	12:	//MoveZ-Free ready? -> Piece zuordnen -> Action ready
		IF NOT pStampSupport^.M_GetActionBusy(E_Action.ACTION_MoveZ) THEN
			nActionState := 80;
			IF bTakePiece THEN
				//Piece von Magazin auf Support übertragen
				IF pStampSupport^.P_bStampInSupport THEN
					//das letze Slot ermitteln
					stError.ErrorId := fbObjectDirectory.M_MoveObject(pPiece,pStampSupport,pStampSupport^.P_nNumberOfSlots);
				ELSE //Take fehlgeschlagen, weil Stamp nicht im Support detektierbar
					stError.ErrorId := E_ErrorIdCmd.ERRORID_PieceExchangeFailed;
				END_IF
			ELSE //Drop
				//Piece von Support auf Magazin übertragen
				IF pStampSupport^.P_bStampInSupport THEN //Drop fehlgeschlagen, weil weil Stamp noch im Support detektierbar
					stError.ErrorId := E_ErrorIdCmd.ERRORID_PieceExchangeFailed;
					nActionState := 99;
				ELSE
					stError.ErrorId := fbObjectDirectory.M_MoveObject(pPiece,pTarget,pPieceSlot^.nNr);
				END_IF
			END_IF
			pPiece^.P_bIgnoreOffset := FALSE;
			IF stError.ErrorId > 0 THEN
				nActionState := 99;
			ELSE
				nActionState := 80;		
			END_IF
		END_IF
		
	70:	//Action abbrechen
		nActionState := 80;
		pPiece^.P_bIgnoreOffset := FALSE;
		IF fbMoveToTarget.bBusy THEN
			fbMoveToTarget(bStop:= TRUE);
			nActionState := 70;
		ELSIF pStampSupport^.M_GetActionBusy(E_Action.ACTION_MoveZ) THEN
			pStampSupport^.M_CancelAction(E_Action.ACTION_MoveZ);
			nActionState := 70;
		ELSE
			fbMoveToTarget(bExecute:= FALSE);
		END_IF
		
		IF pStampSupport^.M_GetActionBusy(E_Action.ACTION_LockUnlock) THEN
			pStampSupport^.M_CancelAction(E_Action.ACTION_LockUnlock);
			nActionState := 70;
		END_IF
		
		IF pStampSupport^.M_GetActionBusy(E_Action.ACTION_StampAdjust) THEN
			pStampSupport^.M_CancelAction(E_Action.ACTION_StampAdjust);
			nActionState := 70;
		END_IF
END_CASE

//Errorhandling
IF nActionState = 99 THEN
	pPiece^.P_bIgnoreOffset := FALSE;
	fbMoveToTarget(bExecute:= FALSE);
	stError.ObjectId := pStampSupport^.P_nObjectID;
	stError.Cmd := E_Action.ACTION_ExchangePiece;
	stError.POUAction := E_POUACT.POUACT_A_ExchangeStamp;
	fbErrorList.M_Add(stError);
END_IF
END_ACTION

ACTION A_ExchangeTip:
stError.POUState := nActionState;

IF pMzTool^.P_bError THEN
	stError.ErrorId := pMzTool^.P_nErrorId;
	nActionState := 99;
END_IF

IF pMzTool^.P_bCanceled AND nActionState > 0 AND nActionState < 70 THEN
	//MzTool wurde durch StopDevice abgebrochen
	nActionState := 70;
END_IF

CASE nActionState OF
	0:	//MoveToTarget auf Slot
		nActionState := 1;
		MEMSET(ADR(stActionData),0,SIZEOF(stActionData));
		stActionData.eAction := E_Action.ACTION_MoveToTarget;
		stActionData.nObject := pMzTool^.P_nObjectID;
		stActionData.nTarget := pTarget^.P_nObjectID;
		stActionData.aParams[1] := E_TargetRef.TARGETREF_Slot;
		stActionData.aParams[2] := pPieceSlot^.nNr;
		stActionData.aParams[3] := 0;
		stActionData.aParams[5] := -1;	//MaxSpeed X
		stActionData.aParams[6] := -1;	//MaxSpeed Y
		stActionData.aParams[7] := -1;	//MaxSpeed Z
		
		IF NOT bTakePiece THEN //Drop
			stDimension :=  pPiece^.P_stDimension;
			stActionData.aParams[10] := - REAL_TO_DINT(stDimension.Height - pPiece^.P_rZOverlapTool);
		END_IF
		
		pPiece^.P_bIgnoreOffset := TRUE;
		
		stError.ErrorId := fbMoveToTarget.M_SetAndCheckParams(stActionData);
		IF stError.ErrorId > 0 THEN	//Error
			nActionState := 99;
		ELSE
			fbMoveToTarget(bExecute:= TRUE);
			nActionState := 1;
		END_IF		
		
	1:	//MoveToTarget ready? -> MoveZ bei Take bzw Eject bei Drop
		fbMoveToTarget(bExecute:= TRUE);
		IF NOT fbMoveToTarget.bBusy THEN
			IF fbMoveToTarget.bError THEN
				stError.ErrorId := fbMoveToTarget.nErrorId;
				nActionState := 99;
			ELSE
				IF bTakePiece THEN //Take
					//Z-Zustellung um OverlapTool und SumDockOffset
					stActionData.eAction := E_Action.ACTION_MoveZ;
					stActionData.aParams[1] := E_MoveMode.MODE_Relative;
					stActionData.aParams[2] := REAL_TO_DINT(pPiece^.P_rZOverlapTool * -1 + rSumDockOffset);
					stActionData.aParams[3] := 4000; //MoveSpeed
				ELSE
					stActionData.eAction := E_Action.ACTION_Eject;
				END_IF
				stError.ErrorId := pMzTool^.M_ExeAction(stActionData);
				IF stError.ErrorId > 0 THEN	//Error
					nActionState := 99;
				ELSE
					nActionState := 2;
				END_IF		
			END_IF
			fbMoveToTarget(bExecute:= FALSE);
		END_IF
		
	2:	//MoveZ bzw Eject ready? -> MoveZ-Home
		IF NOT (pMzTool^.M_GetActionBusy(E_Action.ACTION_MoveZ) OR pMzTool^.M_GetActionBusy(E_Action.ACTION_Eject)) THEN
			nActionState := 3;
			MEMSET(ADR(stActionData),0,SIZEOF(stActionData));
			stActionData.eAction := E_Action.ACTION_MoveZ;
			stActionData.aParams[1] := E_MoveMode.MODE_Home;
			stActionData.aParams[3] := -1; //MoveSpeed
			stError.ErrorId := pMzTool^.M_ExeAction(stActionData);
			IF stError.ErrorId > 0 THEN	//Error
				nActionState := 99;
			END_IF
		END_IF
		
	3:	//MoveZ-Home ready -> Piece zuordnen -> Action ready
		IF NOT pMzTool^.M_GetActionBusy(E_Action.ACTION_MoveZ) THEN
			IF bTakePiece THEN
				//Piece von NeedleRack auf MzTool übertragen
				stError.ErrorId := fbObjectDirectory.M_MoveObject(pPiece,pMzTool,1);
			ELSE
				//Piece von MzTool auf Rack übertragen
				stError.ErrorId := fbObjectDirectory.M_MoveObject(pPiece,pTarget,pPieceSlot^.nNr);
				//Offset von Piece löschen
				stPoint1.X := 0;
				stPoint1.Y := 0;
				stPoint1.Z := 0;
				pPiece^.P_stOffset := stPoint1;
				//Tip als "used" kennzeichnen
				pTip := pPiece;
				pTip^.P_bUsed := TRUE;
				fbObjectDirectory.M_SetObjChange(pPiece^.P_nObjectID);
			END_IF
			pPiece^.P_bIgnoreOffset := FALSE;
			IF stError.ErrorId > 0 THEN
				nActionState := 99;
			ELSE
				nActionState := 80;		
			END_IF
		END_IF
 		
	70:	//Action abbrechen
		pPiece^.P_bIgnoreOffset := FALSE;
		IF fbMoveToTarget.bBusy THEN
			fbMoveToTarget(bStop:= TRUE);
		ELSIF pMzTool^.M_GetActionBusy(E_Action.ACTION_MoveZ) THEN
			pMzTool^.M_CancelAction(E_Action.ACTION_MoveZ);
		ELSE
			fbMoveToTarget(bExecute:= FALSE);
			nActionState := 80;
		END_IF		
END_CASE

//Errorhandling
IF nActionState = 99 THEN
	fbMoveToTarget(bExecute:= FALSE);
	pPiece^.P_bIgnoreOffset := FALSE;
	stError.ObjectId := pMzTool^.P_nObjectID;
	stError.Cmd := E_Action.ACTION_ExchangePiece;
	stError.POUAction := E_POUACT.POUACT_A_ExchangeTip;
	fbErrorList.M_Add(stError);
END_IF
END_ACTION

ACTION A_ExchangeVial:
stError.POUState := nActionState;

IF pMzTool^.P_bError THEN
	stError.ObjectId := pMzTool^.P_nObjectID;
	stError.ErrorId := pMzTool^.P_nErrorId;
	nActionState := 99;
ELSE
	IF pReactor > 0 THEN
		IF pReactor^.P_bError THEN
			stError.ObjectId := pReactor^.P_nObjectID;
			stError.ErrorId := pReactor^.P_nErrorId;
			nActionState := 99;
		END_IF
	END_IF	
END_IF

IF pMzTool^.P_bCanceled AND nActionState > 0 AND nActionState < 70 THEN
	//MzTool wurde durch StopDevice abgebrochen
	nActionState := 70;
END_IF

CASE nActionState OF
	0:	//Prepare
		//Druck
		//Reactor öffnen
		//Überprüfen, ob VialKlemme zu bzw prüfen, ob Vial im Slot
		//VialDetection
		nActionState := 5;
		timer1(IN:= FALSE);
		IF pTarget^.P_eObjectType = E_ObjectType.OBJECTTYPE_Reactor THEN
			pReactor := pTarget;
			MEMSET(ADR(stActionData),0,SIZEOF(stActionData));
			stActionData.eAction := E_Action.ACTION_DetectVial;
			stActionData.aParams[1] := E_OpClState.Open;
			
			stError.ErrorId := pReactor^.M_ExeAction(stActionData);
			IF stError.ErrorId > 0 THEN
				stError.ObjectId := pReactor^.P_nObjectID;
				nActionState := 99;
			ELSE
				nActionState := 1;	
			END_IF			
		END_IF
		
		IF nActionState <> 99 THEN
			//Hier kann die XY-Zustellung bereits angestoßen werden
			MEMSET(ADR(stActionData),0,SIZEOF(stActionData));
			//stActionData.bIntern := TRUE;
			stActionData.eAction := E_Action.ACTION_MoveToTarget;
			stActionData.nObject := pMzTool^.P_nObjectID;
			stActionData.nTarget := pTarget^.P_nObjectID;
			stActionData.aParams[1] := E_TargetRef.TARGETREF_Slot;
			stActionData.aParams[2] := pPieceSlot^.nNr;
			stActionData.aParams[3] := 0;
			stActionData.aParams[5] := -1;	//MaxSpeed X
			stActionData.aParams[6] := -1;	//MaxSpeed Y
			stActionData.aParams[7] := 0;	//MaxSpeed Z
			stError.ErrorId := fbMoveToTarget.M_SetAndCheckParams(stActionData);
			IF stError.ErrorId > 0 THEN	//Error
				stError.ObjectId := pMzTool^.P_nObjectID;
				nActionState := 99;
			ELSE
				IF pMzTool^.P_eObjectType = E_ObjectType.OBJECTTYPE_TriplePip THEN //PneuChannel vorbereiten
					pTriplePip := pMzTool;
					MEMSET(ADR(stActionData),0,SIZEOF(stActionData));
					stActionData.eAction := E_Action.ACTION_SetVacuum;
					IF bTakePiece THEN
						stActionData.aParams[1] := 1; //Fertigmeldung wenn Solldruck erreicht
						stActionData.aParams[2] := -80; //Value in kPa
						stActionData.aParams[3] := 5; //Toleranz
						stActionData.aParams[4] := 5; //Toleranz
						stActionData.aParams[5] := 10000; //Timeout in ms
						stError.ErrorId :=  pMzTool^.M_ExeAction(stActionData);
						IF stError.ErrorId > 0 THEN
							stError.ObjectId := pMzTool^.P_nObjectID;
							nActionState := 99;
						ELSE
							//Ventil aus falls noch an
							MEMSET(ADR(stActionData),0,SIZEOF(stActionData));
							stActionData.eAction := E_Action.ACTION_SwitchPressure;
							stActionData.aParams[1] := E_PressCtrl.PRESSCTRL_Off;
							stError.ErrorId := pMzTool^.M_ExeAction(stActionData);
							IF stError.ErrorId > 0 THEN
								stError.ObjectId := pMzTool^.P_nObjectID;
								nActionState := 99;
							ELSE
								nActionState := 1;
							END_IF
						END_IF
					ELSE
						nActionState := 1;
					END_IF
				END_IF				
			END_IF
		END_IF
		IF nActionState = 1 THEN
			fbMoveToTarget(bExecute:= TRUE);
		END_IF
 		
	1:	//Prepare ready?
		nActionState := 5;
		IF pTarget^.P_eObjectType = E_ObjectType.OBJECTTYPE_Reactor THEN
			nActionState := 2;
			IF pReactor^.M_GetActionBusy(E_Action.ACTION_DetectVial) THEN
				nActionState := 1;
			END_IF
		END_IF
		
		IF pMzTool^.P_eObjectType = E_ObjectType.OBJECTTYPE_TriplePip THEN //Vacuum OK?
			IF pMzTool^.M_GetActionBusy(E_Action.ACTION_SetVacuum) THEN
				nActionState := 1;
			END_IF
		END_IF
		
	2:	//Auswertung VialDetection
		nActionState := 3;
		IF bTakePiece THEN
			IF NOT pReactor^.P_bVialInSlot THEN
				stError.ErrorId := E_ErrorIdCmd.ERRORID_NoVialInReactor;
				nActionState := 99;
			END_IF
		ELSE
			IF pReactor^.P_bVialInSlot THEN
				stError.ErrorId := E_ErrorIdCmd.ERRORID_VialAlreadyInReactor;		
				nActionState := 99;
			END_IF
		END_IF
		
	3:	//Open Reactor
		nActionState := 4;
		MEMSET(ADR(stActionData),0,SIZEOF(stActionData));
		stActionData.eAction := E_Action.ACTION_ReactorOpCl;
		stActionData.aParams[1] := E_ReactDrive.CoverBoth;
		stActionData.aParams[2] := E_OpClCtrl.Open;
		stError.ErrorId := pReactor^.M_ExeAction(stActionData);
		IF stError.ErrorId > 0 THEN
			stError.ObjectId := pReactor^.P_nObjectID;
			nActionState := 99;
		END_IF			
		
	4:	//Reactor open?
		IF NOT pReactor^.M_GetActionBusy(E_Action.ACTION_ReactorOpCl) THEN
			nActionState := 5;
		END_IF
	
	5:	//MoveToTarget Slot
		fbMoveToTarget(bExecute:= TRUE);
		IF NOT fbMoveToTarget.bBusy THEN
			IF fbMoveToTarget.bError THEN
				stError.ErrorId := fbMoveToTarget.nErrorId;
				nActionState := 99;
				fbMoveToTarget(bExecute:= FALSE);
			ELSE
				MEMSET(ADR(stActionData),0,SIZEOF(stActionData));
				stActionData.eAction := E_Action.ACTION_MoveToTarget;
				stActionData.nObject := pMzTool^.P_nObjectID;
				stActionData.nTarget := pTarget^.P_nObjectID;
				stActionData.aParams[1] := E_TargetRef.TARGETREF_Slot;
				stActionData.aParams[2] := pPieceSlot^.nNr;
				stActionData.aParams[3] := 0;
				stActionData.aParams[5] := -1;	//MaxSpeed X
				stActionData.aParams[6] := -1;	//MaxSpeed Y
				stActionData.aParams[7] := -1;	//MaxSpeed Z
				IF bTakePiece THEN
					stActionData.aParams[10] := REAL_TO_DINT(rSumDockOffset);
				END_IF
				fbMoveToTarget(bExecute:= FALSE);
				stError.ErrorId := fbMoveToTarget.M_SetAndCheckParams(stActionData);
				IF stError.ErrorId > 0 THEN	//Error
					stError.ObjectId := pMzTool^.P_nObjectID;
					nActionState := 99;
				ELSE
					fbMoveToTarget(bExecute:= TRUE);
					nActionState := 6;
				END_IF
			END_IF
		END_IF
	
	6:	//MoveToTarget ready? -> Übergabe
		fbMoveToTarget(bExecute:= TRUE);
		IF NOT fbMoveToTarget.bBusy THEN
			IF fbMoveToTarget.bError THEN
				stError.ErrorId := fbMoveToTarget.nErrorId;
				nActionState := 99;
			ELSE
				IF bTakePiece THEN
					nActionState := 7;
				ELSE
					nActionState := 10;
				END_IF
			END_IF
			fbMoveToTarget(bExecute:= FALSE);
		END_IF
		
	7:	//Übergabe Take
		nActionState := 8;
		MEMSET(ADR(stActionData),0,SIZEOF(stActionData));
		stActionData.eAction := E_Action.ACTION_SwitchPressure;
		//Vacuum zuschalten
		stActionData.aParams[1] := E_PressCtrl.PRESSCTRL_VacOn;
		stError.ErrorId := pMzTool^.M_ExeAction(stActionData);
		IF stError.ErrorId > 0 THEN
			stError.ObjectId := pMzTool^.P_nObjectID;
			nActionState := 99;
		END_IF
		
	8:	//Zeit warten
		timer1(IN:= TRUE, PT:=T#1S);
		IF timer1.Q THEN
			timer1(IN:= FALSE);
			nActionState := 9;
		END_IF
		
	9:	//Vaccum OK ? -> MoveZ-Free
		IF pTriplePip^.M_GetVacuumOk(nSetPressValue:= pTriplePip^.P_nHoldVacVial, nSetPressTolPlus:= 0, nSetPressTolMin := 99) THEN
			nActionState := 13;
		END_IF
		
	10:	//Übergabe Drop
		//MoveZ relativ um Slot-Tiefe abzüglich 1mm
		nActionState := 11;
		MEMSET(ADR(stActionData),0,SIZEOF(stActionData));
		stActionData.eAction := E_Action.ACTION_MoveZ;
		stActionData.aParams[1] := E_MoveMode.MODE_Relative;
		stActionData.aParams[2] := -(REAL_TO_DINT((pPieceSlot^.P_rDepth - 1000)));
		stActionData.aParams[3] := 20000; //MoveSpeed
		stError.ErrorId := pMzTool^.M_ExeAction(stActionData);
		IF stError.ErrorId > 0 THEN	//Error
			stError.ObjectId := pMzTool^.P_nObjectID;
			nActionState := 99;
		END_IF
	
	11:	//MoveZ ready? -> MoveX 1mm zum lösen vom Vial, Vacuum Off
		IF NOT pMzTool^.M_GetActionBusy(E_Action.ACTION_MoveZ) THEN
			nActionState := 12;
			//Move 1mm in X, damit Vial sich vom Tool löst
			MEMSET(ADR(stActionData),0,SIZEOF(stActionData));
			stActionData.eAction := E_Action.ACTION_MoveX;
			stActionData.aParams[1] := E_MoveMode.MODE_Relative;
			stActionData.aParams[2] := 500;
			stActionData.aParams[3] := 10000; //MoveSpeed
			stActionData.aParams[4] := 1; //Ignore Collision
			stError.ErrorId := pMzTool^.M_ExeAction(stActionData);
			IF stError.ErrorId > 0 THEN	//Error
				stError.ObjectId := pMzTool^.P_nObjectID;
				nActionState := 99;
			ELSE
				//Vacuum OFF
				MEMSET(ADR(stActionData),0,SIZEOF(stActionData));
				stActionData.eAction := E_Action.ACTION_SwitchPressure;
				stActionData.aParams[1] := E_PressCtrl.PRESSCTRL_Off;
				stError.ErrorId :=  pMzTool^.M_ExeAction(stActionData);
				IF stError.ErrorId > 0 THEN
					stError.ObjectId := pMzTool^.P_nObjectID;
					nActionState := 99;
				ELSE
					//Set Vacuum "0"
					MEMSET(ADR(stActionData),0,SIZEOF(stActionData));
					stActionData.eAction := E_Action.ACTION_SetVacuum;
					stActionData.aParams[1] := 0; //Fertigmeldung sofort
					stActionData.aParams[2] := 0; //Value in kPa
					stError.ErrorId :=  pMzTool^.M_ExeAction(stActionData);
					IF stError.ErrorId > 0 THEN
						stError.ObjectId := pMzTool^.P_nObjectID;
						stError.POUState := nActionState;
						nActionState := 99;
					END_IF
				END_IF
			END_IF
		END_IF
		
	12:	//MoveX ready? -> MoveZ 1mm nach oben
		IF NOT pMzTool^.M_GetActionBusy(E_Action.ACTION_MoveX) THEN
			nActionState := 13;
			MEMSET(ADR(stActionData),0,SIZEOF(stActionData));
			stActionData.eAction := E_Action.ACTION_MoveZ;
			stActionData.aParams[1] := E_MoveMode.MODE_Relative;
			stActionData.aParams[2] := 500; //0,5mm nach oben
			stActionData.aParams[3] := 1000; //MoveSpeed
			stError.ErrorId :=  pMzTool^.M_ExeAction(stActionData);
			IF stError.ErrorId > 0 THEN
				stError.ObjectId := pMzTool^.P_nObjectID;
				nActionState := 99;
			END_IF
		END_IF
		
	13:	//MoveZ-Free
		IF NOT pMzTool^.M_GetActionBusy(E_Action.ACTION_MoveZ) THEN
			MEMSET(ADR(stActionData),0,SIZEOF(stActionData));
			stActionData.eAction := E_Action.ACTION_MoveZ;
			stActionData.aParams[1] := E_MoveMode.MODE_Home;
			stActionData.aParams[3] := -1; //MoveSpeed
			stError.ErrorId := pMzTool^.M_ExeAction(stActionData);
			IF stError.ErrorId > 0 THEN	//Error
				stError.ObjectId := pMzTool^.P_nObjectID;
				nActionState := 99;
			END_IF
			nActionState := 14;
		END_IF

	14:	//MoveZ-Free ready? -> Action ready
		IF NOT pMzTool^.M_GetActionBusy(E_Action.ACTION_MoveZ) THEN
			IF bTakePiece THEN	//Vial von Target auf MzTool übertragen
				stError.ErrorId := fbObjectDirectory.M_MoveObject(pPiece,pMzTool,1);
				pVial := pPiece;
				pVial^.P_bUsed := TRUE;
				fbObjectDirectory.M_SetObjChange(pPiece^.P_nObjectID);
			ELSE	//Vial von MzTool auf Target übertragen
				stError.ErrorId := fbObjectDirectory.M_MoveObject(pPiece,pTarget,pPieceSlot^.nNr);
			END_IF
			IF stError.ErrorId > 0 THEN
				nActionState := 99;
			ELSE
				nActionState := 80;		
			END_IF
		END_IF
		
	70:	//Abbrechen
		IF NOT bTakePiece THEN
			nActionState := 71;
		ELSE
			nActionState := 80;
		END_IF
	
		IF fbMoveToTarget.bBusy THEN
			fbMoveToTarget(bStop:= TRUE);
			nActionState := 70;
		ELSIF pMzTool^.M_GetActionBusy(E_Action.ACTION_MoveX) THEN
			pMzTool^.M_CancelAction(E_Action.ACTION_MoveX);
			nActionState := 70;
		ELSIF pMzTool^.M_GetActionBusy(E_Action.ACTION_MoveZ) THEN
			pMzTool^.M_CancelAction(E_Action.ACTION_MoveZ);
			nActionState := 70;
		END_IF
		
		IF pMzTool^.M_GetActionBusy(E_Action.ACTION_SetVacuum) THEN
			nActionState := 70;
			pMzTool^.M_CancelAction(E_Action.ACTION_SetVacuum);
		END_IF
		
		IF pMzTool^.M_GetActionBusy(E_Action.ACTION_SwitchPressure) THEN
			nActionState := 70;
			pMzTool^.M_CancelAction(E_Action.ACTION_SwitchPressure);
		END_IF
		
		IF pReactor > 0 THEN
			IF pReactor^.M_GetActionBusy(E_action.ACTION_ReactorOpCl) THEN
				pReactor^.M_CancelAction(E_action.ACTION_ReactorOpCl);
				nActionState := 70;
			ELSIF pReactor^.M_GetActionBusy(E_action.ACTION_DetectVial) THEN
				pReactor^.M_CancelAction(E_action.ACTION_DetectVial);
				nActionState := 70;
			END_IF
		END_IF	
	
	71:	//Vacuum OFF (nur wenn Take)
		nActionState := 80;
		stActionData.eAction := E_Action.ACTION_SwitchPressure;
		stActionData.aParams[1] := E_PressCtrl.PRESSCTRL_Off;
		stError.ErrorId := pMzTool^.M_ExeAction(stActionData);
		IF stError.ErrorId = 0 THEN
			stActionData.eAction := E_Action.ACTION_SetVacuum;
			stActionData.aParams[1] := 0; //Sofortige Fertigmeldung
			stActionData.aParams[2] := 0; //Druck
			stError.ErrorId := pMzTool^.M_ExeAction(stActionData);
			IF stError.ErrorId > 0 THEN
				stError.ObjectId := pMzTool^.P_nObjectID;
				nActionState := 99;
			END_IF
		END_IF	
END_CASE

//Errorhandling
IF nActionState = 99 THEN
	IF bTakePiece THEN
		stActionData.eAction := E_Action.ACTION_SwitchPressure;
		stActionData.aParams[1] := E_PressCtrl.PRESSCTRL_Off;
		pMzTool^.M_ExeAction(stActionData);
		stActionData.eAction := E_Action.ACTION_SetVacuum;
		stActionData.aParams[1] := 0; //Sofortige Fertigmeldung
		stActionData.aParams[2] := 0; //Druck
		pMzTool^.M_ExeAction(stActionData);
	END_IF
	pPiece^.P_bIgnoreOffset := FALSE;
	fbMoveToTarget(bExecute:= FALSE);
	stError.ObjectId := pMzTool^.P_nObjectID;
	stError.Cmd := E_Action.ACTION_ExchangePiece;
	stError.POUAction := E_POUACT.POUACT_A_ExchangeVial;
	fbErrorList.M_Add(stError);
END_IF
END_ACTION

ACTION A_ExchangeVialGripper:
stError.POUState := nActionState;

IF pMzTool^.P_bError THEN
	stError.ObjectId := pMzTool^.P_nObjectID;
	stError.ErrorId := pMzTool^.P_nErrorId;
	nActionState := 99;
ELSE
	IF pPowderStation > 0 AND_THEN pTarget = pPowderStation THEN
		IF pPowderStation^.P_bError THEN
			stError.ObjectId := pPowderStation^.P_nObjectID;
			stError.ErrorId := pPowderStation^.P_nErrorId;
			nActionState := 99;
		END_IF
	ELSIF pReactor > 0 AND_THEN pTarget = pReactor THEN
		IF pReactor^.P_bError THEN
			stError.ObjectId := pReactor^.P_nObjectID;
			stError.ErrorId := pReactor^.P_nErrorId;
			nActionState := 99;
		END_IF
	END_IF
END_IF

IF pMzTool^.P_bCanceled AND nActionState > 0 AND nActionState < 70 THEN
	//MzTool wurde durch StopDevice abgebrochen
	nActionState := 70;
END_IF

CASE nActionState OF
	0:	//Move free für Gripper-Test
		MEMSET(ADR(stActionData),0,SIZEOF(stActionData));
		stActionData.eAction := E_Action.ACTION_MoveZ;
		stActionData.aParams[1] := E_MoveMode.MODE_Home;
		stActionData.aParams[3] := -1; //MoveSpeed
		stError.ErrorId := pMzTool^.M_ExeAction(stActionData);
		IF stError.ErrorId > 0 THEN	//Error
			stError.ObjectId := pMzTool^.P_nObjectID;
			nActionState := 99;
		ELSE
			nActionState := 1;
		END_IF
		
	1:	//Move free ready?
		IF NOT pMzTool^.M_GetActionBusy(E_Action.ACTION_MoveZ) THEN
			//Gripper vorbereiten bzw. checken, ob State zur Belegung des VialSlots passt.
			//Auch bei TakePiece muss zuerst geschlosse werden, da ja aus irgendwelchen Gründen
			//noch ein Vial im Greifer sein kann und das Vial womöglich auf die Workplate falle würde
			stError.ErrorId := pGripper^.M_OpenClose(E_OpClCtrl.Close, FALSE);
			IF stError.ErrorId = 0 THEN
				nActionState := 2;
			ELSE
				nActionState := 99;
			END_IF			
		END_IF
	
	2:	//Gripper ready?
		IF NOT pGripper^.M_GetActionBusy(E_Action.ACTION_OpenClose) THEN
			IF bTakePiece THEN
				//Muss vollständig geschlossen sein, was bedeutet, dass sich kein Vial im Gripper befindet
				IF pGripper^.P_eCurrentGripperState = E_GripperState.FullyClosed THEN
					//wieder öffnen
					stError.ErrorId := pGripper^.M_OpenClose(E_OpClCtrl.Open, FALSE);
					IF stError.ErrorId = 0 THEN
						nActionState := 3;
					ELSE
						nActionState := 99;	
					END_IF
				ELSE
					stError.ErrorId := E_ErrorIdCmd.ERRORID_ToolNotFreeOrBlocked;
					nActionState := 99;
				END_IF
			ELSE //Drop
				IF pGripper^.P_eCurrentGripperState = E_GripperState.HalfClosed THEN
					IF pTarget^.P_eObjectType = E_ObjectType.OBJECTTYPE_PowderStation THEN
						nActionState := 10;
					 	
					ELSIF pTarget^.P_eObjectType = E_ObjectType.OBJECTTYPE_Reactor THEN
						nActionState := 20;
					ELSE
						nActionState := 30;
					END_IF
				ELSE
					stError.ErrorId := E_ErrorIdCmd.ERRORID_NoPieceOnTool;
					nActionState := 99;
				END_IF
			END_IF
		END_IF
		
	3:	//Gripper ready?
		IF NOT pGripper^.M_GetActionBusy(E_Action.ACTION_OpenClose) THEN
			IF pGripper^.P_eCurrentGripperState = E_GripperState.Open THEN
				IF pTarget^.P_eObjectType = E_ObjectType.OBJECTTYPE_PowderStation THEN
					nActionState := 10;
				ELSIF pTarget^.P_eObjectType = E_ObjectType.OBJECTTYPE_Reactor THEN
					nActionState := 20;
				ELSE
					nActionState := 30;
				END_IF
 			ELSE
				stError.ErrorId := E_ErrorIdCmd.ERRORID_CouldNotOpenGripper;
				nActionState := 99;
			END_IF
		END_IF
		
	10:	//PowderStation in ReloadPos fahren
		stActionData.eAction := E_Action.ACTION_PowdStatReload;
		stError.ErrorId := pPowderStation^.M_ExeAction(stActionData);
		IF stError.ErrorId > 0 THEN	//Error
			stError.ObjectId := pPowderStation^.P_nObjectID;
			nActionState := 99;
		ELSE
			nActionState := 11;
		END_IF
		
	11:	//RealoadPos ready?
		IF NOT pPowderStation^.M_GetActionBusy(E_Action.ACTION_PowdStatReload) THEN
			nActionState := 30;
		END_IF
		
	20: //Reaktor ist noch nicht implementiert
		stError.ErrorId := E_ErrorIdCmd.ERRORID_InvalidTarget;
		nActionState := 99;
		
	30:	//Wenn Drop, dann muss noch über den Vialdetector überprüft werden,
		//ob nicht schon ein Vial im Target steckt. Dazu muss also ein MoveToTarget
		//mit entsprechendem Offset gemacht werden.
		IF bTakePiece THEN
			nActionState := 32;
		ELSE
			//move zur Übergabe mit Offset und checken
			MEMSET(ADR(stActionData),0,SIZEOF(stActionData));
			stActionData.eAction := E_Action.ACTION_MoveToTarget;
			stActionData.nObject := pMzTool^.P_nObjectID;
			stActionData.nTarget := pTarget^.P_nObjectID;
			stActionData.aParams[1] := E_TargetRef.TARGETREF_Slot;
			stActionData.aParams[2] := pPieceSlot^.nNr;
			stActionData.aParams[3] := 0;
			stActionData.aParams[5] := -1;	//MaxSpeed X
			stActionData.aParams[6] := -1;	//MaxSpeed Y
			stActionData.aParams[7] := -1;	//MaxSpeed Z
			stActionData.aParams[8] :=	0;	//Offset X
			stActionData.aParams[9] :=	-25500;	//Offset Y
			stActionData.aParams[10] :=	15000;	//Offset Z	
			stError.ErrorId := fbMoveToTarget.M_SetAndCheckParams(stActionData);
			IF stError.ErrorId > 0 THEN	//Error
				stError.ObjectId := pMzTool^.P_nObjectID;
				nActionState := 99;
			ELSE
				fbMoveToTarget(bExecute:= TRUE);
				nActionState := 31;
			END_IF
		END_IF
	
	31:	//MoveToTarget ready?
		fbMoveToTarget();
		IF NOT fbMoveToTarget.bBusy THEN
			IF fbMoveToTarget.bError THEN
				stError.ErrorId := fbMoveToTarget.nErrorId;
				nActionState := 99;
			ELSE
				IF NOT pGripper^.P_bVialDetector THEN //Es befindet sich ein Vial im Target
					stError.ErrorId := E_ErrorIdCmd.ERRORID_PieceAlreadyInSlot;
					nActionState := 99;
				ELSE
					//Eigentlicher MoveToTarget
					nActionState := 32;
				END_IF
			END_IF
			fbMoveToTarget(bExecute:= FALSE);
		END_IF
		
	32:	//MoveToTarget
		MEMSET(ADR(stActionData),0,SIZEOF(stActionData));
		stActionData.eAction := E_Action.ACTION_MoveToTarget;
		stActionData.nObject := pMzTool^.P_nObjectID;
		stActionData.nTarget := pTarget^.P_nObjectID;
		stActionData.aParams[1] := E_TargetRef.TARGETREF_Slot;
		stActionData.aParams[2] := pPieceSlot^.nNr;
		stActionData.aParams[3] := 0;
		stActionData.aParams[5] := -1;	//MaxSpeed X
		stActionData.aParams[6] := -1;	//MaxSpeed Y
		stActionData.aParams[7] := 30000;	//Speed Z
		IF bTakePiece THEN
			stActionData.aParams[10] := -REAL_TO_DINT(pPiece^.P_rZOverlapTool);
		END_IF
		
		stError.ErrorId := fbMoveToTarget.M_SetAndCheckParams(stActionData);
		IF stError.ErrorId > 0 THEN	//Error
			stError.ObjectId := pMzTool^.P_nObjectID;
			nActionState := 99;
		ELSE
			fbMoveToTarget(bExecute:= TRUE);
			nActionState := 33;
		END_IF
	
	33:	//MoveToTarget ready?
		fbMoveToTarget();
		IF NOT fbMoveToTarget.bBusy THEN
			IF fbMoveToTarget.bError THEN
				stError.ErrorId := fbMoveToTarget.nErrorId;
				nActionState := 99;
			ELSE
				IF bTakePiece THEN
					nActionState := 40;
				ELSE //Drop
					nActionState := 42;
				END_IF
			END_IF
			fbMoveToTarget(bExecute:= FALSE);
		END_IF
		
	40:	//Übergabe Take -> Close Gripper
		stError.ErrorId := pGripper^.M_OpenClose(E_OpClCtrl.Close, FALSE);
		IF stError.ErrorId > 0 THEN
			nActionState := 99;
		ELSE
			nActionState := 41;
		END_IF
		
	41:	//Gripper closed? (HALF)
		IF NOT pGripper^.M_GetActionBusy(E_Action.ACTION_OpenClose) THEN
			IF pGripper^.P_eCurrentGripperState = E_GripperState.HalfClosed THEN
				nActionState := 50; //Move free
			ELSE
				stError.ErrorId := E_ErrorIdCmd.ERRORID_NoPieceTaken;
				nActionState := 99;
			END_IF
		END_IF
		
	42:	//Übergabe Drop ->MoveZ relativ um Slot-Tiefe abzüglich 1mm
		MEMSET(ADR(stActionData),0,SIZEOF(stActionData));
		stActionData.eAction := E_Action.ACTION_MoveZ;
		stActionData.aParams[1] := E_MoveMode.MODE_Relative;
		stActionData.aParams[2] := -(REAL_TO_DINT((pPieceSlot^.P_rDepth - 1000)));
		stActionData.aParams[3] := 20000; //MoveSpeed
		stError.ErrorId := pMzTool^.M_ExeAction(stActionData);
		IF stError.ErrorId > 0 THEN	//Error
			stError.ObjectId := pMzTool^.P_nObjectID;
			nActionState := 99;
		ELSE
			nActionState := 43;
		END_IF
		
	43: //MoveZ ready? -> Open Gripper
		IF NOT pMzTool^.M_GetActionBusy(E_Action.ACTION_MoveZ) THEN
			stError.ErrorId := pGripper^.M_OpenClose(E_OpClCtrl.Open, FALSE);
			IF stError.ErrorId > 0 THEN
				nActionState := 99;
			ELSE
				nActionState := 44;
			END_IF
		END_IF
		
	44:	//Gripper open?
		IF NOT pGripper^.M_GetActionBusy(E_Action.ACTION_OpenClose) THEN
			IF pGripper^.P_eCurrentGripperState = E_GripperState.Open THEN
				nActionState := 50; //Move free
			ELSE
				stError.ErrorId := E_ErrorIdCmd.ERRORID_NotFullyOpened;
				nActionState := 99;
			END_IF
		END_IF
		
	50:	//Move free
		MEMSET(ADR(stActionData),0,SIZEOF(stActionData));
		stActionData.eAction := E_Action.ACTION_MoveZ;
		stActionData.aParams[1] := E_MoveMode.MODE_Home;
		stActionData.aParams[3] := -1; //MoveSpeed
		stError.ErrorId := pMzTool^.M_ExeAction(stActionData);
		IF stError.ErrorId > 0 THEN	//Error
			stError.ObjectId := pMzTool^.P_nObjectID;
			nActionState := 99;
		ELSE
			nActionState := 51;
		END_IF
		
	51:	//MoveZ-Free ready? -> Action ready
		IF NOT pMzTool^.M_GetActionBusy(E_Action.ACTION_MoveZ) THEN
			//Vial richtig angekommen? Geht nur bei Gripper, Reaktor oder bei PowderStation
			IF bTakePiece THEN
				IF pGripper^.P_eCurrentGripperState = E_GripperState.HalfClosed THEN
					nActionState := 60; //weiter zu Vial im OD verschieben
				ELSE
					stError.ErrorId := E_ErrorIdCmd.ERRORID_NoPieceTaken;
					nActionState := 99;
				END_IF
			ELSE //Drop
				IF pTarget^.P_eObjectType = E_ObjectType.OBJECTTYPE_Reactor THEN
					//Hier muss die DetectAction noch ausgeführt werden
					MEMSET(ADR(stActionData),0,SIZEOF(stActionData));
					stActionData.eAction := E_Action.ACTION_DetectVial;
					stActionData.aParams[1] := E_OpClState.Closed;
					stError.ErrorId := pReactor^.M_ExeAction(stActionData);
					IF stError.ErrorId > 0 THEN
						stError.ObjectId := pReactor^.P_nObjectID;
						nActionState := 99;
					ELSE
						//nActionState := 15; //Überprüfung, ob Vial auch im Reaktor angekommen???
					END_IF
				ELSE
					nActionState := 60; //weiter zu Vial im OD verschieben
				END_IF
			END_IF
		END_IF
		
	60:	//Vial im OD verschieben
		IF bTakePiece THEN	//Vial von Target auf MzTool übertragen
			stError.ErrorId := fbObjectDirectory.M_MoveObject(pPiece,pMzTool,1);
			pVial := pPiece;
			//pVial^.P_bUsed := TRUE;
			fbObjectDirectory.M_SetObjChange(pPiece^.P_nObjectID);
		ELSE	//Vial von MzTool auf Target übertragen
			stError.ErrorId := fbObjectDirectory.M_MoveObject(pPiece,pTarget,pPieceSlot^.nNr);
		END_IF
		IF stError.ErrorId > 0 THEN
			nActionState := 99;
		ELSE
			nActionState := 80;		
		END_IF
	
	70:	//Abbrechen
		nActionState := 80;
		
		IF fbMoveToTarget.bBusy THEN
			fbMoveToTarget(bStop:= TRUE);
			nActionState := 70;
		ELSIF pMzTool^.M_GetActionBusy(E_Action.ACTION_MoveX) THEN
			pMzTool^.M_CancelAction(E_Action.ACTION_MoveX);
			nActionState := 70;
		ELSIF pMzTool^.M_GetActionBusy(E_Action.ACTION_MoveZ) THEN
			pMzTool^.M_CancelAction(E_Action.ACTION_MoveZ);
			nActionState := 70;
		END_IF
		
		IF pReactor > 0 THEN
			IF pReactor^.M_GetActionBusy(E_action.ACTION_ReactorOpCl) THEN
				pReactor^.M_CancelAction(E_action.ACTION_ReactorOpCl);
				nActionState := 70;
			ELSIF pReactor^.M_GetActionBusy(E_action.ACTION_DetectVial) THEN
				pReactor^.M_CancelAction(E_action.ACTION_DetectVial);
				nActionState := 70;
			END_IF
		END_IF	

END_CASE

//Errorhandling
IF nActionState = 99 THEN
	pPiece^.P_bIgnoreOffset := FALSE;
	fbMoveToTarget(bExecute:= FALSE);
	stError.ObjectId := pMzTool^.P_nObjectID;
	stError.Cmd := E_Action.ACTION_ExchangePiece;
	stError.POUAction := E_POUACT.POUACT_A_ExchangeVialGripper;
	fbErrorList.M_Add(stError);
END_IF
END_ACTION

ACTION A_GetPipSample:
stError.POUState := nActionState;

IF pMzTool^.P_bError THEN
	stError.ObjectId := pMzTool^.P_nObjectID;
	stError.ErrorId := pMzTool^.P_nErrorId;
	nActionState := 99;
END_IF

IF pMzTool^.P_bCanceled AND nActionState > 0 AND nActionState < 70 THEN
	//MzTool wurde durch StopDevice abgebrochen
	nActionState := 70;
END_IF

CASE nActionState OF
	0:	//MoveToTarget zu Mtp in PrePos
		timer1(IN:= FALSE);
		MEMSET(ADR(stActionData),0,SIZEOF(stActionData));
		stActionData.eAction := E_Action.ACTION_MoveToTarget;
		IF pMzTool^.P_eObjectType = E_ObjectType.OBJECTTYPE_TwinPiezoHolder THEN
			stActionData.nObject := pTwinPiezoHolder^.P_pPiezoPipFirst^.P_nObjectID;
		ELSE
			stActionData.nObject := pMzTool^.P_nObjectID;	
		END_IF
		stActionData.nTarget := pMtp^.P_nObjectID;
		stActionData.aParams[1] := E_TargetRef.TARGETREF_TwoDimArray;
		stActionData.aParams[2] := nCol;
		stActionData.aParams[3] := nRow;
		stActionData.aParams[5] := -1;	//MaxSpeed X
		stActionData.aParams[6] := -1;	//MaxSpeed Y
		stActionData.aParams[7] := -1;	//MaxSpeed Z
		stError.ErrorId := fbMoveToTarget.M_SetAndCheckParams(stActionData);
		IF stError.ErrorId > 0 THEN
			stError.ObjectId := pMzTool^.P_nObjectID;
			nActionState := 99;
		ELSE
			fbMoveToTarget(bExecute:= TRUE);
			nActionState := 1;
		END_IF
		
	1:	//MoveToTarget ready?
		fbMoveToTarget(bExecute:= TRUE);
		IF NOT fbMoveToTarget.bBusy THEN
			IF fbMoveToTarget.bError THEN
				stError.ErrorId := fbMoveToTarget.nErrorId;
				nActionState := 99;
			ELSE
				IF nQuantity2 > 0 THEN //AirGap
					MEMSET(ADR(stActionData),0,SIZEOF(stActionData));
					stActionData.eAction := E_Action.ACTION_Aspirate;
					stActionData.aParams[1] := nQuantity2; //Quantity Airgap
					stActionData.aParams[2] := nFlow1;
					stError.ErrorId := pMzTool^.M_ExeAction(stActionData);
					IF stError.ErrorId > 0 THEN
						nActionState := 99;
					ELSE
						nActionState := 2;
					END_IF
				ELSE
					nActionState := 4;
				END_IF
			END_IF
			fbMoveToTarget(bExecute:= FALSE);
		END_IF	
		
	2: //AirGap ready?
		IF NOT pMzTool^.M_GetActionBusy(E_Action.ACTION_Aspirate) THEN
			IF nTime > 0 THEN
				timer1(IN:= TRUE, PT:= DWORD_TO_TIME(nTime));
				nActionState := 3;
			ELSE
				nActionState := 4;
			END_IF
		END_IF
		
	3:	//Delay elapsed?
		timer1();
		IF timer1.Q THEN
			timer1(IN:= FALSE);
			nActionState := 4;
		END_IF
	
	4:	//Eintauchen in Well
		stPoint1 := pMtp^.M_GetAbsPos(pChildPos:= 0, eTargetRef:= E_TargetRef.TARGETREF_TwoDimArray, nParam1:= nCol, nParam2:= nRow,
									nParam3:= 1,nZLevel:= 1);			
		MEMSET(ADR(stActionData),0,SIZEOF(stActionData));
		stActionData.eAction := E_Action.ACTION_MoveZ;
		stActionData.aParams[1] := E_MoveMode.MODE_AbsWithOffset;
		stActionData.aParams[2] := REAL_TO_DINT(stPoint1.Z);
		stActionData.aParams[3] := -1;
		stError.ErrorId := pMzTool^.M_ExeAction(stActionData);
		IF stError.ErrorId > 0 THEN
			stError.ObjectId := pMzTool^.P_nObjectID;
			nActionState := 99;
		ELSE
			nActionState := 5;	
		END_IF
		
	5:	//Eintauchen ready? -> Aspirieren
		IF NOT pMzTool^.M_GetActionBusy(E_Action.ACTION_MoveZ) THEN
			nActionState := 6;
			MEMSET(ADR(stActionData),0,SIZEOF(stActionData));
			stActionData.eAction := E_Action.ACTION_Aspirate;
			stActionData.aParams[1] := nQuantity1;
			stActionData.aParams[2] := nFlow1;
			stError.ErrorId := pMzTool^.M_ExeAction(stActionData);
			IF stError.ErrorId > 0 THEN
				stError.ObjectId := pMzTool^.P_nObjectID;
				stError.POUState := nActionState;
				nActionState := 99;
			ELSE
				IF bGetPipSample_ActivatePiezo THEN
					MEMSET(ADR(stActionData),0,SIZEOF(stActionData));
					stActionData.eAction := E_Action.ACTION_DispenseDrops;
					stActionData.aParams[2] := 1; //Ein
					stActionData.aParams[5] := 1; //Skip valve move
					pMzTool^.M_ExeAction(stActionData);
				END_IF
			END_IF
		END_IF
		
	6:	//Aspirate ready? -> Delay
		IF NOT pMzTool^.M_GetActionBusy(E_Action.ACTION_Aspirate) THEN
			IF nTime > 0 THEN
				timer1(IN:= TRUE, PT:= DWORD_TO_TIME(nTime));
				nActionState := 7;
			ELSE
				nActionState := 8;
			END_IF
		END_IF
	
	7:	//Delay elapsed? -> bei Piezo au Bypass sonst MoveZ_Free
		timer1();
		IF timer1.Q THEN
			timer1(IN:= FALSE);
			IF pMzTool^.P_eObjectType = E_ObjectType.OBJECTTYPE_PiezoPip THEN
				nActionState := 8;
			ELSE
				nActionState := 10;
			END_IF
		END_IF
		
	8:	//Valve auf Bypass stellen
		IF bGetPipSample_SwitchBypass THEN
			MEMSET(ADR(stActionData),0,SIZEOF(stActionData));
			stActionData.eAction := E_Action.ACTION_DilMoveValve;
			stActionData.aParams[1] := 3; //Bypass-Position
			stError.ErrorId := pMzTool^.M_ExeAction(stActionData);
			IF stError.ErrorId > 0 THEN
				nActionState := 99;
			ELSE
				nActionState := 9;	
			END_IF		
		ELSE
			nActionState := 10;
		END_IF
		
	9:	//Valve auf Bypass?
		IF NOT pMzTool^.M_GetActionBusy(E_Action.ACTION_DilMoveValve) THEN
			nActionState := 10;
		END_IF
	
	10:	//MoveZ-Free
		pMzTool^.M_CancelAction(E_Action.ACTION_DispenseDrops);
		MEMSET(ADR(stActionData),0,SIZEOF(stActionData));
		stActionData.eAction := E_Action.ACTION_MoveZ;
		stActionData.aParams[1] := E_MoveMode.MODE_Free;
		stActionData.aParams[3] := -1; //MaxSpeed Z
		stError.ErrorId := pMzTool^.M_ExeAction(stActionData);
		IF stError.ErrorId > 0 THEN
			stError.ObjectId := pMzTool^.P_nObjectID;
			nActionState := 99;
		ELSE
			nActionState := 11;
		END_IF
		
	11:	//MoveZ-Free ready?
		IF NOT pMzTool^.M_GetActionBusy(E_Action.ACTION_MoveZ) THEN
			nActionState := 80;
 		END_IF
		
	70:	//Abbrechen
		nActionState := 80;
		IF fbMoveToTarget.bBusy THEN
			fbMoveToTarget(bStop:= TRUE);
			nActionState := 70;
		ELSIF pMzTool^.M_GetActionBusy(E_Action.ACTION_MoveZ) THEN
			pMzTool^.M_CancelAction(E_Action.ACTION_MoveZ);
			nActionState := 70;
		ELSE
			fbMoveToTarget(bExecute := FALSE);
		END_IF
		
		IF pMzTool^.M_GetActionBusy(E_Action.ACTION_Aspirate) THEN
			pMzTool^.M_CancelAction(E_Action.ACTION_Aspirate);
			nActionState := 70;
		END_IF
		
		IF pMzTool^.M_GetActionBusy(E_Action.ACTION_DilMoveValve) THEN
			pMzTool^.M_CancelAction(E_Action.ACTION_DilMoveValve);
			nActionState := 70;
		END_IF
END_CASE

//Errorhandling
IF nActionState = 99 THEN
	fbMoveToTarget(bExecute:= FALSE);
	stError.Cmd := E_Action.ACTION_GetPipSample;
	stError.ObjectId := pMzTool^.P_nObjectID;
	stError.POUAction := E_POUACT.POUACT_A_GetPipSample;
	fbErrorList.M_Add(stError);
END_IF
END_ACTION

ACTION A_InsertTool:
stError.POUState := nActionState;

IF pMzTool^.P_bError THEN
	stError.ErrorId := pMzTool^.P_nErrorId;
	nActionState := 99;
END_IF

IF pMzTool^.P_bCanceled AND nActionState > 0 AND nActionState < 70 THEN
	//MzTool wurde durch StopDevice abgebrochen
	nActionState := 70;
END_IF

CASE nActionState OF
	0:	//MoveToTarget auf Slot
		//Wenn aktuelle XY-Position des Tools mit der Position des Slots übereinstimmt(Tolerenz +-5µm)
		//muss kann MoveToTarget übersprungen werden
		//Hilfreich beim Anheben der Needle auf anderes Level ohne dass vorher herausgezogen wird
		stPoint1 := pMzTool^.P_stCurrentPosPhys;
		stPoint2 := pTarget^.M_GetAbsPos(pChildPos:= 0, eTargetRef,nTargetCol,nTargetRow,0,0);
		IF ABS(stPoint1.X - stPoint2.X) <= 5.0 AND ABS(stPoint1.Y - stPoint2.Y) <= 5.0 THEN
			nActionState := 3; //-> EIntauchen
			RETURN;
		END_IF
 		
		MEMSET(ADR(stActionData),0,SIZEOF(stActionData));
		stActionData.eAction := E_Action.ACTION_MoveToTarget;
		stActionData.nObject := pMzTool^.P_nObjectID;
		stActionData.nTarget := pTarget^.P_nObjectID;
		stActionData.aParams[1] := eTargetRef;
		stActionData.aParams[2] := nTargetCol;
		stActionData.aParams[3] := nTargetRow;
		stActionData.aParams[5] := -1;	//MaxSpeed X
		stActionData.aParams[6] := -1;	//MaxSpeed Y
		stActionData.aParams[7] := -1;	//MaxSpeed Z
		IF pTarget^.P_eObjectType = E_ObjectType.OBJECTTYPE_FlipTubeRack THEN
			stActionData.aParams[8] := -4000;	//XOffset	
			stActionData.aParams[10] := 1000;	//ZOffset	
		END_IF
		
		stError.ErrorId := fbMoveToTarget.M_SetAndCheckParams(stActionData);
		IF stError.ErrorId > 0 THEN	//Error
			nActionState := 99;
		ELSE
			fbMoveToTarget(bExecute:= TRUE);
			nActionState := 1;
		END_IF		
		
	1:	//MoveToTarget ready? (nur für FlipTube) (Deckel etwas weiter öffnen) MoveX
		fbMoveToTarget(bExecute:= TRUE);
		IF NOT fbMoveToTarget.bBusy THEN
			IF fbMoveToTarget.bError THEN
				stError.ErrorId := fbMoveToTarget.nErrorId;
				nActionState := 99;
			ELSE
				IF pTarget^.P_eObjectType = E_ObjectType.OBJECTTYPE_FlipTubeRack THEN //MoveX (Deckel öffnen)
					MEMSET(ADR(stActionData),0,SIZEOF(stActionData));
					stActionData.eAction := E_Action.ACTION_MoveX;
					stActionData.aParams[1] := E_MoveMode.MODE_Relative;
					stActionData.aParams[2] := 13000;
					stActionData.aParams[3] := 45000;
					stActionData.aParams[4] := 1;
					stError.ErrorId := pMzTool^.M_ExeAction(stActionData);
					IF stError.ErrorId > 0 THEN	//Error
						nActionState := 99;
					ELSE
						nActionState := 2;	
					END_IF
				ELSE	//Eintauchen
					nActionState := 4;
				END_IF
			END_IF
			fbMoveToTarget(bExecute:= FALSE);
		END_IF
		
	2:	//MoveX ready? (nur für FlipTube) (zur Mitte zurück)
		IF NOT pMzTool^.M_GetActionBusy(E_Action.ACTION_MoveX) THEN
			MEMSET(ADR(stActionData),0,SIZEOF(stActionData));
			stActionData.eAction := E_Action.ACTION_MoveX;
			stActionData.aParams[1] := E_MoveMode.MODE_Relative;
			stActionData.aParams[2] := -9000; 
			stActionData.aParams[3] := 45000;
			stActionData.aParams[4] := 1;
			stError.ErrorId := pMzTool^.M_ExeAction(stActionData);
			IF stError.ErrorId > 0 THEN	//Error
				nActionState := 99;
			ELSE
				nActionState := 3;
			END_IF
		END_IF
		
	3:	IF NOT pMzTool^.M_GetActionBusy(E_Action.ACTION_MoveX) THEN
			nActionState := 4;
		END_IF

	4:	//Eintauchen
		//Eintauchen bis InsertLevel
		MEMSET(ADR(stActionData),0,SIZEOF(stActionData));
		stActionData.eAction := E_Action.ACTION_MoveZ;
		stActionData.aParams[1] := E_MoveMode.MODE_AbsWithOffset;;
		stActionData.aParams[3] := 10000; //Speed (wird ev. überschrieben durch reduzierte Eintauchgeschwindigkeit
		
		IF eTargetRef = E_TargetRef.TARGETREF_Slot THEN
			stPoint1 := pTarget^.M_GetAbsPos(pChildPos:= 0, eTargetRef,nTargetCol,0,0,0);
			IF pPieceSlot^.P_pPiece > 0 THEN
				IF pPieceSlot^.P_pPiece^.P_eObjectType = E_ObjectType.OBJECTTYPE_Vial OR pPieceSlot^.P_pPiece^.P_eObjectType = E_ObjectType.OBJECTTYPE_VialClosed THEN
					pVial := pPieceSlot^.P_pPiece;
					IF nInsertLevel = 0 THEN
						stActionData.aParams[2] := REAL_TO_DINT(stPoint1.Z) + pVial^.P_nTopLevel;
						pMzTool^.P_nReducedMoveZDist := - pVial^.P_nTopLevel;
					ELSE
						stActionData.aParams[2] := REAL_TO_DINT(stPoint1.Z) + pVial^.P_nBottomLevel;
						pMzTool^.P_nReducedMoveZDist := - pVial^.P_nBottomLevel;
					END_IF
					IF pVial^.P_eObjectType = E_ObjectType.OBJECTTYPE_VialClosed OR pMzTool^.P_eObjectType = E_ObjectType.OBJECTTYPE_TitrationTool THEN
						stActionData.aParams[3] := 10000;
						pMzTool^.P_nReducedMoveZSpeed := 10000;
					END_IF
				ELSIF pPieceSlot^.P_pPiece^.P_eObjectType = E_ObjectType.OBJECTTYPE_FlipTube THEN
					pFlipTube := pPieceSlot^.P_pPiece;
					IF nInsertLevel = 0 THEN
						stActionData.aParams[2] := REAL_TO_DINT(stPoint1.Z) + pFlipTube^.P_nTopLevel;
					ELSE
						stActionData.aParams[2] := REAL_TO_DINT(stPoint1.Z) + pFlipTube^.P_nBottomLevel;
					END_IF
				END_IF
			END_IF
		ELSIF eTargetRef = E_TargetRef.TARGETREF_TwoDimArray THEN
			stPoint1 := pTarget^.M_GetAbsPos(pChildPos:= 0, eTargetRef,nTargetCol,nTargetRow,0, nInsertLevel);
			stActionData.aParams[2] := REAL_TO_DINT(stPoint1.Z);
		END_IF
		
		stError.ErrorId := pMzTool^.M_ExeAction(stActionData);
		IF stError.ErrorId > 0 THEN	//Error
			nActionState := 99;
		ELSE
			nActionState := 5;
		END_IF			
		
	5:	//MoveZ ready? -> Action ready
		IF NOT pMzTool^.M_GetActionBusy(E_Action.ACTION_MoveZ) THEN
			nActionState := 80;
		END_IF
		
	70:	//Abbrechen
		IF fbMoveToTarget.bBusy THEN
			fbMoveToTarget(bStop:= TRUE);
		ELSE
			IF pMzTool^.M_GetActionBusy(E_Action.ACTION_MoveX) THEN
				pMzTool^.M_CancelAction(E_Action.ACTION_MoveX);
			ELSIF pMzTool^.M_GetActionBusy(E_Action.ACTION_MoveZ) THEN
				pMzTool^.M_CancelAction(E_Action.ACTION_MoveZ);
			ELSE
				fbMoveToTarget(bExecute:= FALSE);
				nActionState := 80;
			END_IF
		END_IF
END_CASE

//Errorhandling
IF nActionState = 99 THEN
	fbMoveToTarget(bExecute:= FALSE);
	stError.ObjectId := pMzTool^.P_nObjectID;
	stError.Cmd := E_Action.ACTION_InsertTool;
	stError.POUAction := E_POUACT.POUACT_A_InsertTool;
	fbErrorList.M_Add(stError);
END_IF
END_ACTION

ACTION A_MeasureStamp:
stError.POUState := nActionState;

IF pMzTool^.P_bError THEN
	stError.ObjectId := pMzTool^.P_nObjectID;
	stError.ErrorId := pMzTool^.P_nErrorId;
	nActionState := 99;
END_IF

IF pMzTool^.P_bCanceled AND nActionState > 0 AND nActionState < 70 THEN
	//MzTool wurde durch StopDevice abgebrochen
	nActionState := 70;
END_IF

CASE nActionState OF
	0:	//MoveToTarget auf "MeasurePoint"
		pStampSupport := pMzTool;
		pPiece := pStampSupport^.P_pPiece;
		pPiece^.P_bIgnoreOffset := FALSE;
		
		MEMSET(ADR(stActionData),0,SIZEOF(stActionData));
		stActionData.eAction := E_Action.ACTION_MoveToTarget;
		stActionData.nObject := pStampSupport^.P_nObjectID;
		stActionData.nTarget := pTarget^.P_nObjectID;
		stActionData.aParams[1] := E_TargetRef.TARGETREF_SpecPoint;
		stActionData.aParams[2] := 1; //MeasurePoint
		stActionData.aParams[5] := -1;	//MaxSpeed X
		stActionData.aParams[6] := -1;	//MaxSpeed Y
		stActionData.aParams[7] := -1;	//Speed Z
		stActionData.aParams[10] := 9000;	//ZOffset
		stError.ErrorId := fbMoveToTarget.M_SetAndCheckParams(stActionData);
		IF stError.ErrorId > 0 THEN	//Error
			nActionState := 99;
		ELSE
			fbMoveToTarget(bExecute:= TRUE);
			nActionState := 1;
		END_IF
		
	1:	//MoveToTarget ready?
		fbMoveToTarget(bExecute:= TRUE);
		IF NOT fbMoveToTarget.bBusy THEN
			IF fbMoveToTarget.bError THEN
				stError.ErrorId := fbMoveToTarget.nErrorId;
			ELSE
				nActionState := 2;	
			END_IF
			fbMoveToTarget(bExecute:= FALSE);
		END_IF
	
	2:	//MoveZ langsam (max 5mm) nach unten bis Sensor schaltet
		nActionState := 3;
		MEMSET(ADR(stActionData),0,SIZEOF(stActionData));
		stActionData.eAction := E_Action.ACTION_MoveZ;
		stActionData.aParams[1] := E_MoveMode.MODE_Relative;
		stActionData.aParams[2] := -12000;
		stActionData.aParams[3] := 2000;
		stError.ErrorId := pStampSupport^.M_ExeAction(stActionData);
		IF stError.ErrorId > 0 THEN	//Error
			nActionState := 99;
		END_IF
	
	3:	//MoveZ ready oder Sensor -> MoveZ Stop
		IF iTargetZSensor.P_bSensor THEN
			pStampSupport^.M_CancelAction(E_Action.ACTION_MoveZ);
			IF NOT pStampSupport^.M_GetActionBusy(E_Action.ACTION_MoveZ) THEN
				nActionState := 4;
			END_IF
		ELSE
			IF NOT pStampSupport^.M_GetActionBusy(E_Action.ACTION_MoveZ) THEN
				//Sensor not reached -> Sensor defect
				stError.ErrorId := E_ErrorIdCmd.ERRORID_MeasureZDistanceExeeded;
				nActionState := 99;
			END_IF
		END_IF
	
	4:	//MoveZ langsam (max 5mm) nach oben bis Sensor schaltet
		nActionState := 5;
		MEMSET(ADR(stActionData),0,SIZEOF(stActionData));
		//stActionData.bIntern := TRUE;
		stActionData.eAction := E_Action.ACTION_MoveZ;
		stActionData.aParams[1] := E_MoveMode.MODE_Relative;
		stActionData.aParams[2] := 3000;
		stActionData.aParams[3] := 200;
		stError.ErrorId := pStampSupport^.M_ExeAction(stActionData);
		IF stError.ErrorId > 0 THEN	//Error
			nActionState := 99;
		END_IF
	
	5:	//Warten bis MoveZ fertig bzw Sensor schaltet
		IF NOT iTargetZSensor.P_bSensor THEN
			pStampSupport^.M_CancelAction(E_Action.ACTION_MoveZ);
		END_IF
		
		IF NOT pStampSupport^.M_GetActionBusy(E_Action.ACTION_MoveZ) THEN
			nActionState := 6;
		ELSIF NOT pStampSupport^.M_GetActionBusy( E_Action.ACTION_MoveZ) THEN
			stError.ErrorId := E_ErrorIdCmd.ERRORID_MeasureZDistanceExeeded;
			nActionState := 99;
		END_IF
		
	6:	//MoveZ-Free und ZOffset eintragen
		nActionState := 7; 
		stMeasCalibPoint := pTarget^.M_GetAbsPos(pChildPos:= 0, E_TargetRef.TARGETREF_SpecPoint,1,0,0, nZLevel:=0);
		stMeasCurrentPos := pStampSupport^.P_stCurrentPosPhys;
		stMeasOffset := pPiece^.P_stOffset;
		stMeasOffset.Z := stMeasOffset.Z + stMeasCalibPoint.Z - stMeasCurrentPos.Z;
		pPiece^.P_stOffset := stMeasOffset; 
  		
		fbObjectDirectory.M_SetObjChange(pPiece^.P_nObjectID);

		//Freifahren
		MEMSET(ADR(stActionData),0,SIZEOF(stActionData));
		//stActionData.bIntern := TRUE;
		stActionData.eAction := E_Action.ACTION_MoveZ;
		stActionData.aParams[1] := E_MoveMode.MODE_Free;
		stActionData.aParams[3] := -1; //MaxSpeed Z
		stError.ErrorId := pStampSupport^.M_ExeAction(stActionData);
		IF stError.ErrorId > 0 THEN	//Error
			nActionState := 99;
		END_IF
		
	7:	//MoveZ-Free ready? -> Action ready
		IF NOT pStampSupport^.M_GetActionBusy( E_Action.ACTION_MoveZ)  THEN
			nActionState := 80;
		END_IF
		
	70:	//Abbrechen
		//MoveToTarget oder MoveZ vom MzTool abbrechen (schließen sich gegenseitig aus)
		IF fbMoveToTarget.bBusy THEN
			fbMoveToTarget(bStop:= TRUE);
		ELSIF pMzTool^.M_GetActionBusy(E_Action.ACTION_MoveZ) THEN
			pMzTool^.M_CancelAction(E_Action.ACTION_MoveZ);
		ELSE
			fbMoveToTarget(bExecute:= FALSE);			
			nActionState := 80;
		END_IF
END_CASE

//Errorhandling
IF nActionState = 99 THEN
	fbMoveToTarget(bExecute:= FALSE);
	stError.ObjectId := pMzTool^.P_nObjectID;
	stError.Cmd := E_Action.ACTION_MeasureTool;
	stError.POUAction := E_POUACT.POUACT_A_MeasureStamp;
	fbErrorList.M_Add(stError);
END_IF
END_ACTION

ACTION A_MeasureTarget:
stError.POUState := nActionState;

IF pMzTool^.P_bError THEN
	stError.ErrorId := pMzTool^.P_nErrorId;
	nActionState := 99;
END_IF

IF pMzTool^.P_bCanceled AND nActionState > 1 AND nActionState < 70 THEN
	//MzTool wurde durch StopDevice abgebrochen
	nActionState := 70;
END_IF

CASE nActionState OF
	0:	//Z-SensorID auslesen
		fbReadZSensorID(pFbZAxisRef:= pMzTool^.P_pZAxisRef, bExecute := TRUE);
		IF NOT fbReadZSensorID.bBusy THEN
			IF fbReadZSensorID.bError THEN
				stError.ErrorId := fbReadZSensorID.nErrorID;
				nActionState := 99;
			ELSE
				nZSensorId := pMzTool^.P_pZAxisRef^.P_nZSensorID;
				//Z-SensorCalibrationValue ermitteln
				rZSensorCalibration := pMzTool^.P_pFbMultiZ^.M_GetZSensorCalib(nZSensorId,pMzTool^.P_nZAxisNr);
				IF rZSensorCalibration = 0.0 THEN //Error
					stError.ErrorId := ERRORID_ZSensorNotCalibrated;
					nActionState := 99;
				ELSE
					//TargetPosition ermitteln
					IF eMeasTipOption = E_MeasureOption.MEAS_OPTION_SlowApproach THEN
						pTarget^.P_rZOffset := 0;
						fbObjectDirectory.M_SetObjChange(pTarget^.P_nObjectID);
					END_IF
					//Bei Inkstation wird nur SpecPoint2 vermessen
					IF pTarget^.P_eObjectType = E_ObjectType.OBJECTTYPE_InkStation THEN
						stMeasureTargetTgtPos := pTarget^.M_GetAbsPos(pChildPos:= 0, eTargetRef:= E_TargetRef.TARGETREF_SpecPoint,
																		nParam1:= 2,
																		nParam2:= 0,
																		nParam3:= 0,
																		nZLevel:= 0);
					ELSE
						stMeasureTargetTgtPos := pTarget^.P_stAbsPosCenter;	
					END_IF
					nActionState := 1;
				END_IF				
			END_IF
			fbReadZSensorID(bExecute := FALSE);
		END_IF

	1:	//Wenn Mode "Auto" dann in MoveXY zu TargetPos
		IF eMeasureTargetMode = E_MeasureMode.MEAS_MODE_Auto THEN
			nActionState := 2;
			//Move XY zum Target
			MEMSET(ADR(stActionData),0,SIZEOF(stActionData));
			stActionData.eAction := E_Action.ACTION_MoveXY;
			stActionData.aParams[1] := E_MoveMode.MODE_AbsWithOffset;
			stActionData.aParams[2] := REAL_TO_DINT(stMeasureTargetTgtPos.X); //XPos
			stActionData.aParams[3] := REAL_TO_DINT(stMeasureTargetTgtPos.Y); //YPos
			stActionData.aParams[4] := -1;	//MaxSpeed X
			stActionData.aParams[5] := -1;	//MaxSpeed Y
			stError.ErrorId := pMzTool^.M_ExeAction(stActionData);
			IF stError.ErrorId > 0 THEN	//Error
				nActionState := 99;
			END_IF
		END_IF
		
	2:	//MoveXY ready? -> MoveZ PrePos
		IF NOT pMzTool^.M_GetActionBusy(E_Action.ACTION_MoveXY) THEN
			nActionState := 3;
			IF eMeasTipOption = E_MeasureOption.MEAS_OPTION_FastApproach THEN
				MEMSET(ADR(stActionData),0,SIZEOF(stActionData));
				stActionData.eAction := E_Action.ACTION_MoveZ;
				stActionData.aParams[1] := E_MoveMode.MODE_AbsWithOffset;
				stActionData.aParams[2] := REAL_TO_DINT(stMeasureTargetTgtPos.Z) + 5000; 
				stActionData.aParams[3] := -1; //MaxSpeed Z
				stError.ErrorId := pMzTool^.M_ExeAction(stActionData);
				IF stError.ErrorId > 0 THEN	//Error
					nActionState := 99;
				END_IF
			END_IF
		END_IF
		
	3:	//MoveZ ready? start Measurement 
		IF NOT pMzTool^.M_GetActionBusy(E_Action.ACTION_MoveZ) THEN
			nActionState := 4;
			MEMSET(ADR(stActionData),0,SIZEOF(stActionData));
			stActionData.eAction := E_Action.ACTION_MoveZ;
			stActionData.aParams[1] := E_MoveMode.MODE_Measure;
			stMeasCurrentPos := pMzTool^.P_stCurrentPosTotal;
			rMeasureTargetDistance := stMeasureTargetTgtPos.Z - stMeasCurrentPos.Z - 4500;
			stActionData.aParams[2] := REAL_TO_DINT(rMeasureTargetDistance);
			stActionData.aParams[3] := 10000;	//Speed nur damit kein Fehler von MultiZ auftritt(MeasureSpeed ist fix)
			stError.ErrorId := pMzTool^.M_ExeAction(stActionData);
			IF stError.ErrorId > 0 THEN	//Error
				nActionState := 99;
			END_IF
		END_IF
		
	4:	//Measurement ready? -> Offsets berechnen, MoveZ-Free
		IF NOT pMzTool^.M_GetActionBusy(E_Action.ACTION_MoveZ) THEN
			nActionState := 5;
			//Neue Gesamthöhe = CalibrationValue - AktAxisPos(Raw)
			stPoint1.Z := pMzTool^.P_pZAxisRef^.P_rCurrentPos - rZSensorCalibration;
			//Differenz aus alter Gesamthöhe und neuer Gesamthöhe ermitteln
			stPoint2.Z := stPoint1.Z - stMeasureTargetTgtPos.Z;
			//Diese Differnz auf Offset des Targets aufschlagen
			pTarget^.P_rZOffset := pTarget^.P_rZOffset + stPoint2.Z;
			//MoveZ-Free		
			MEMSET(ADR(stActionData),0,SIZEOF(stActionData));
			//stActionData.bIntern := TRUE;
			stActionData.eAction := E_Action.ACTION_MoveZ;
			stActionData.aParams[1] := E_MoveMode.MODE_Home;
			stActionData.aParams[3] := -1; //MaxSpeedZ
			stError.ErrorId := pMzTool^.M_ExeAction(stActionData);
			IF stError.ErrorId > 0 THEN	//Error
				nActionState := 99;
			END_IF	
		END_IF
		
	5:	//MoveZ-Free ready? -> Action ready
		IF NOT pMzTool^.M_GetActionBusy(E_Action.ACTION_MoveZ) THEN
			fbObjectDirectory.M_SetObjChange(pTarget^.P_nObjectID);
			nActionState := 80;
		END_IF

	70:	//Action abbrechen
		IF fbReadZSensorID.bBusy THEN
			fbReadZSensorID(bExecute:= FALSE);
		ELSIF pMzTool^.M_GetActionBusy(E_Action.ACTION_MoveXY) THEN
			pMzTool^.M_CancelAction(E_Action.ACTION_MoveXY);
		ELSIF pMzTool^.M_GetActionBusy(E_Action.ACTION_MoveZ) THEN
			pMzTool^.M_CancelAction(E_Action.ACTION_MoveZ);
		ELSE
			nActionState := 80;
		END_IF
		
END_CASE

//Errorhandling
IF nActionState = 99 THEN
	fbMoveToTarget(bExecute:= FALSE);
	stError.ObjectId := pMzTool^.P_nObjectID;
	stError.Cmd := E_Action.ACTION_MeasureTool;
	stError.POUAction := E_POUACT.POUACT_A_MeasureTarget;
	fbErrorList.M_Add(stError);
END_IF
END_ACTION

ACTION A_MeasureTip:
stError.POUState := nActionState;

IF pMzTool^.P_bError THEN
	stError.ErrorId := pMzTool^.P_nErrorId;
	nActionState := 99;
END_IF

CASE nActionState OF
	0:	//Alle Achsen des Heads auf Home fahren
		MEMSET(ADR(stActionData),0,SIZEOF(stActionData));
		stActionData.eAction := E_Action.ACTION_MoveZ;
		stActionData.aParams[1] := E_MoveMode.MODE_Home;
		stActionData.aParams[3] := -1;	//MaxSpeed Z
		stError.ErrorId := pMzTool^.P_pMzHead^.M_ExeAction(stActionData);
		IF stError.ErrorId > 0 THEN
			nActionState := 99;
		ELSE
			nActionState := 1;
		END_IF
		
	1:	//Head ready?
		IF NOT pMzTool^.P_pMzHead^.M_GetActionBusy(E_Action.ACTION_MoveZ) THEN
			IF pMzTool^.P_pMzHead^.P_bError THEN
				stError.ErrorId := pMzTool^.P_pMzHead^.P_nErrorId;
				nActionState := 99;
			ELSE
				nActionState := 2;
			END_IF
		END_IF
		
	2:	//Wenn noch nicht vermessen wurde und angeforderte Option = "MEAS_OPTION_OnlyXY", dann
		//Option auf "MEAS_OPTION_SlowApproach" ändern
		stPoint1 := pMzTool^.P_stRelPos;
		stPoint2 := pMzTool^.P_stOffset;
		
		IF (NOT pMzTool^.P_bMeasured AND eMeasTipOption = E_MeasureOption.MEAS_OPTION_OnlyXY) OR (stPoint1.Z = 0 AND stPoint2.Z = 0) THEN
			eMeasTipOption := E_MeasureOption.MEAS_OPTION_SlowApproach;
		END_IF
		
		IF eMeasTipOption = E_MeasureOption.MEAS_OPTION_SlowApproach THEN
			IF pMzTool^.pPiece > 0 THEN
				pMzTool^.pPiece^.M_ClearOffset();
			ELSE
				pMzTool^.M_ClearOffset();	
			END_IF
		END_IF
		
		//Berechnung Startpos X-Direction
		stMeasPassIntersect := pTipCalibrator^.M_GetAbsPos(pChildPos:= 0, eTargetRef:= E_TargetRef.TARGETREF_SpecPoint,nParam1:= 1, nParam2:=0, nParam3:=0, nZLevel:=0);
		stMeasCalibPoint := pTipCalibrator^.M_GetAbsPos(pChildPos:= 0, eTargetRef:= E_TargetRef.TARGETREF_SpecPoint,nParam1:= 2, nParam2:=0, nParam3:=0, nZLevel:=0);
		stMeasStartPos := stMeasPassIntersect;
		stMeasStartPos.X := stMeasStartPos.X + rMeasureDistance;
		stMeasEndPos := stMeasPassIntersect;
		stMeasEndPos.X := stMeasEndPos.X - rMeasureDistance;
		//MoveXY		
		MEMSET(ADR(stActionData),0,SIZEOF(stActionData));
		stActionData.eAction := E_Action.ACTION_MoveXY;
		stActionData.aParams[1] := E_MoveMode.MODE_AbsWithOffset;
		stActionData.aParams[2] := REAL_TO_DINT(stMeasStartPos.X); //XPos
		stActionData.aParams[3] := REAL_TO_DINT(stMeasStartPos.Y); //YPos
		stActionData.aParams[4] := -1;	//MaxSpeed X
		stActionData.aParams[5] := -1;	//MaxSpeed Y
		
		nActionState := 20;	//Execute MoveAction
		nActionStateNext := 3; //danach weiter zu Z-Zustellung
	
	3:	//MoveZ
		MEMSET(ADR(stActionData),0,SIZEOF(stActionData));
		stActionData.eAction := E_Action.ACTION_MoveZ;
		stActionData.aParams[1] := E_MoveMode.MODE_AbsWithOffset;
		stActionData.aParams[3] := -1;	//MaxSpeed Z
		//In Abhängigkeit von MeasOption "Z" zustellen und Z-Feed voreinstellen
		CASE eMeasTipOption OF
			E_MeasureOption.MEAS_OPTION_SlowApproach: //keine Z-Zustellung, es von oben angefangen
				fbMeasTip.nZFeedStart := -1000;
				fbMeasTip.nZFeedEnde := -25;
				nActionState := 4; //weiter zu Z-Measurement
			E_MeasureOption.MEAS_OPTION_FastApproach:
				stActionData.aParams[1] := E_MoveMode.MODE_AbsWithOffset;
				fbMeasTip.nZFeedStart := -1000;
				fbMeasTip.nZFeedEnde := -25;
				fbMeasTip.nZFeedMax := -4000;
				stActionData.aParams[2] := REAL_TO_DINT(stMeasStartPos.Z); //ZPos
				nActionState := 20; //Execute MoveAction
				nActionStateNext := 4;	//danach weiter zu Z-Measurement
			E_MeasureOption.MEAS_OPTION_OnlyXY:
				stActionData.aParams[1] := E_MoveMode.MODE_AbsWithOffset;		
				stActionData.aParams[2] := REAL_TO_DINT(stMeasCalibPoint.Z) -300; //ZPos
				nActionState := 20; //Execute MoveAction
				nActionStateNext := 7;	//danach weiter zu X-Measurement
		ELSE
			stError.ErrorId := E_ErrorIdCmd.ERRORID_InvalidMeasureMode;
		END_CASE
		bFlag := TRUE;
		
	4:	//Z-Measurement
		IF bFlag THEN
			bFlag := FALSE;
			//FeedMax (maximaler Gesamtvorschub Z berechnen
			IF eMeasTipOption = E_MeasureOption.MEAS_OPTION_SlowApproach THEN
				stPoint1 := pMzTool^.P_stCurrentPosPhys;
				IF pMzTool^.P_pPiece > 0 THEN
					stDimension := pMzTool^.P_pPiece^.P_stDimension;
					stPoint2 := pTarget^.P_stAbsPosCenter;
					fbMeasTip.nZFeedMax := -(REAL_TO_DINT(stPoint1.Z - stPoint2.Z + stDimension.Height - pMzTool^.P_pPiece^.P_rZOverlapTool))- 5000;
				ELSE
					stPoint2 := pTarget^.M_GetAbsPos(pChildPos:= 0, E_TargetRef.TARGETREF_SpecPoint,2,0,0,0); //CalibPoint
					fbMeasTip.nZFeedMax := -(REAL_TO_DINT(stPoint1.Z - stPoint2.Z + 5500));
				END_IF
			END_IF
			
			IF NOT pTipCalibrator^.P_bXSensor THEN
				stError.ErrorId := E_ErrorIdCmd.ERRORID_TipCalibProbeSensorX;
				nActionState := 99;
			END_IF
		END_IF
		
		IF nActionState <> 99 THEN
		fbMeasTip(bExecute:= TRUE, pMzTool:= pMzTool, pTipCalibrator:= pTipCalibrator, nDirection:= 3,
					 stStartPos:= stMeasStartPos, stEndPos:= stMeasEndPos);
		
			IF NOT fbMeasTip.bBusy THEN
				IF fbMeasTip.bError THEN //Error
					stError.ErrorId := fbMeasTip.nErrorId;
					nActionState := 99;
				ELSE
					//Gemessenen Z Wert verrechnen und als OffsetWert in Tool bzw Piece eintragen
					IF pMzTool^.pPiece > 0 THEN
						stMeasOffset := pMzTool^.pPiece^.P_stOffset;
						stMeasOffset.Z := stMeasOffset.Z - (fbMeasTip.stProbePos.Z - stMeasCalibPoint.Z);
						stMeasOffset.X := stMeasOffset.X - (fbMeasTip.stProbePos.X - stMeasCalibPoint.X);
						pMzTool^.pPiece^.P_stOffset := stMeasOffset;
					ELSE
						stMeasOffset := pMzTool^.P_stOffset;
						stMeasOffset.Z := stMeasOffset.Z - (fbMeasTip.stProbePos.Z - stMeasCalibPoint.Z);
						stMeasOffset.X := stMeasOffset.X - (fbMeasTip.stProbePos.X - stMeasCalibPoint.X);
						pMzTool^.P_stOffset := stMeasOffset;
					END_IF
					
					//Berechnung Startpos Y-Direction
					stMeasStartPos := stMeasPassIntersect;
					//für Vermessung HT-Extruder, der in Y-Vermessung teilweise in Y-Min-Limit fährt
					stXYLimits := pMzTool^.M_GetXYRange();
					stMeasStartPos.Y := MAX((stMeasStartPos.Y - rMeasureDistance),stXYLimits.Y1 + 1.000);
					/////////////////////////////////////////////////////////////////////////////////
					stMeasEndPos := stMeasPassIntersect;
					stMeasEndPos.Y := stMeasEndPos.Y + rMeasureDistance;
					//MoveXY		
					MEMSET(ADR(stActionData),0,SIZEOF(stActionData));
					stActionData.eAction := E_Action.ACTION_MoveXY;
					stActionData.aParams[1] := E_MoveMode.MODE_AbsWithOffset;
					stActionData.aParams[2] := REAL_TO_DINT(stMeasStartPos.X); //XPos
					stActionData.aParams[3] := REAL_TO_DINT(stMeasStartPos.Y); //YPos
					stActionData.aParams[4] := -1;	//MaxSpeed X
					stActionData.aParams[5] := -1;	//MaxSpeed Y
					stActionData.aParams[6] := 1;	//Disable crash check
					
					nActionState := 20;		//Execute MoveAction
					nActionStateNext := 5;	//danach weiter zu MoveZ 300µ below CalibPoint
				END_IF
				fbMeasTip(bExecute:= FALSE);	
			END_IF
		END_IF

	5:	//MoveZ
		MEMSET(ADR(stActionData),0,SIZEOF(stActionData));
		stActionData.eAction := E_Action.ACTION_MoveZ;
		stActionData.aParams[1] := E_MoveMode.MODE_AbsWithOffset;
		stActionData.aParams[2] := REAL_TO_DINT(stMeasCalibPoint.Z) -300;
		stActionData.aParams[3] := -1;	//MaxSpeed Z
		nActionStateNext := 6;	//danach weiter zu Y-Measurement
		nActionState := 20; //Execute MoveAction	
	
	6:	//Y-Measurement
		IF bFlag THEN
			bFlag := FALSE;
			IF NOT pTipCalibrator^.P_bYSensor THEN
				stError.ErrorId := E_ErrorIdCmd.ERRORID_TipCalibProbeSensorY;
			END_IF
		END_IF
	
		fbMeasTip(bExecute:= TRUE, pMzTool:= pMzTool, pTipCalibrator:= pTipCalibrator, nDirection:= 2,
					stStartPos:= stMeasStartPos, stEndPos:= stMeasEndPos);		
	
		IF NOT fbMeasTip.bBusy THEN
			IF fbMeasTip.bError THEN
				stError.ErrorId := fbMeasTip.nErrorId;
				nActionState := 99;
			ELSE
				//Gemessenen Y Wert verrechnen und als OffsetWert in Tool eintragen
				IF pMzTool^.pPiece > 0 THEN
					stMeasOffset := pMzTool^.pPiece^.P_stOffset;
					stMeasOffset.Y := stMeasOffset.Y - (fbMeasTip.stProbePos.Y - stMeasCalibPoint.Y);
					pMzTool^.pPiece^.P_stOffset := stMeasOffset;
				ELSE
					stMeasOffset := pMzTool^.P_stOffset;
					stMeasOffset.Y := stMeasOffset.Y - (fbMeasTip.stProbePos.Y - stMeasCalibPoint.Y);
					pMzTool^.P_stOffset := stMeasOffset;
				END_IF
				
				IF eMeasTipOption = E_MeasureOption.MEAS_OPTION_OnlyXY THEN	//Freifahren, denn X wurde bereits durch Z-Measurement erledigt
					MEMSET(ADR(stActionData),0,SIZEOF(stActionData));
					stActionData.eAction := E_Action.ACTION_MoveZ;
					stActionData.aParams[1] := E_MoveMode.MODE_Free;
					stActionData.aParams[3] := -1;	//MaxSpeed Z
					nActionState := 20;
					nActionStateNext := 80;	//Ready!				
				ELSE
					//Berechnung Startpos X-Direction
					stMeasStartPos := stMeasPassIntersect;
					stMeasStartPos.X := stMeasStartPos.X + rMeasureDistance;
					stMeasEndPos := stMeasPassIntersect;
					stMeasEndPos.X := stMeasEndPos.X - rMeasureDistance;
					//MoveXY		
					MEMSET(ADR(stActionData),0,SIZEOF(stActionData));
					stActionData.eAction := E_Action.ACTION_MoveXY;
					stActionData.aParams[1] := E_MoveMode.MODE_AbsWithOffset;
					stActionData.aParams[2] := REAL_TO_DINT(stMeasStartPos.X); //XPos
					stActionData.aParams[3] := REAL_TO_DINT(stMeasStartPos.Y); //YPos
					stActionData.aParams[4] := -1;	//MaxSpeed X
					stActionData.aParams[5] := -1;	//MaxSpeed Y
					stActionData.aParams[6] := 1;	//Disable crash check
					
					nActionState := 20;		//Execute MoveAction
					nActionStateNext := 7;	//danach weiter zu X-Measurement
				END_IF
			END_IF
			fbMeasTip(bExecute:= FALSE);	
		END_IF	
	
	7:	//X-Measurement
		IF bFlag THEN
			bFlag := FALSE;
			IF NOT pTipCalibrator^.P_bXSensor THEN
				stError.ErrorId := E_ErrorIdCmd.ERRORID_TipCalibProbeSensorX;
			END_IF
		END_IF
	
		fbMeasTip(bExecute:= TRUE, pMzTool:= pMzTool, pTipCalibrator:= pTipCalibrator, nDirection:= 1,
					stStartPos:= stMeasStartPos, stEndPos:= stMeasEndPos);
					
		IF NOT fbMeasTip.bBusy THEN
			IF fbMeasTip.bError THEN
				stError.ErrorId := fbMeasTip.nErrorId;
			ELSE
				//Wenn Piece am Tool, den Offset des Pieces verrechnen sonst des Tools
				IF pMzTool^.pPiece > 0 THEN
					stMeasOffset := pMzTool^.pPiece^.P_stOffset;
					stMeasOffset.X := stMeasOffset.X - (fbMeasTip.stProbePos.X - stMeasCalibPoint.X);
					pMzTool^.pPiece^.P_stOffset := stMeasOffset;
				ELSE
					stMeasOffset := pMzTool^.P_stOffset;
					stMeasOffset.X := stMeasOffset.X - (fbMeasTip.stProbePos.X - stMeasCalibPoint.X);
					pMzTool^.P_stOffset := stMeasOffset;
				END_IF
				
				MEMSET(ADR(stActionData),0,SIZEOF(stActionData));
				IF eMeasTipOption = E_MeasureOption.MEAS_OPTION_OnlyXY THEN
					//Berechnung Startpos Y-Direction
					stMeasStartPos := stMeasPassIntersect;
					//für Vermessung HT-Extruder, der in Y-Vermessung teilweise in Y-Min-Limit fährt
					stXYLimits := pMzTool^.M_GetXYRange();
					stMeasStartPos.Y := MAX((stMeasStartPos.Y - rMeasureDistance),stXYLimits.Y1 + 1.000);
					/////////////////////////////////////////////////////////////////////////////////
					stMeasEndPos := stMeasPassIntersect;
					stMeasEndPos.Y := stMeasEndPos.Y + rMeasureDistance;
					//MoveXY		
					stActionData.eAction := E_Action.ACTION_MoveXY;
					stActionData.aParams[1] := E_MoveMode.MODE_AbsWithOffset;
					stActionData.aParams[2] := REAL_TO_DINT(stMeasStartPos.X); //XPos
					stActionData.aParams[3] := REAL_TO_DINT(stMeasStartPos.Y); //YPos
					stActionData.aParams[4] := -1;	//MaxSpeed X
					stActionData.aParams[5] := -1;	//MaxSpeed Y
					stActionData.aParams[6] := 1;	//Disable crash check
					
					nActionState := 20;		//Execute MoveAction
					nActionStateNext := 6;	//danach weiter zu Y-Measurement
				ELSE
					//MoveZ-Free
					stActionData.eAction := E_Action.ACTION_MoveZ;
					stActionData.aParams[1] := E_MoveMode.MODE_Free;
					stActionData.aParams[3] := -1;	//MaxSpeed Z
					
					nActionState := 20;		//Execute MoveAction
					nActionStateNext := 80;	//Ready
					pMzTool^.P_bMeasured := TRUE;
				END_IF
			END_IF
			fbMeasTip(bExecute:= FALSE);
		END_IF						
END_CASE

CASE nActionState OF
	20:	//Execute Move-Action
		stError.ErrorId := pMzTool^.M_ExeAction(stActionData);
		nActionState := 21;
		IF stError.ErrorId > 0 THEN
			nActionState := 99;
		END_IF
	
	21:	//Move-Action ready? ready?
		IF NOT pMzTool^.M_GetActionBusy(stActionData.eAction) THEN
			nActionState := nActionStateNext;
			bFlag := TRUE;
			IF nActionState = 80 THEN
				IF pMzTool^.P_pPiece > 0 THEN
					fbObjectDirectory.M_SetObjChange(pMzTool^.pPiece^.P_nObjectID);
				ELSE
					fbObjectDirectory.M_SetObjChange(pMzTool^.P_nObjectID);
				END_IF
			END_IF
		END_IF
		
	70:	//Action abbrechen
		nActionState := 80;
		IF fbMeasTip.bBusy THEN
			fbMeasTip.M_Cancel();
			fbMeasTip();
			nActionState := 70;
		ELSE
			fbMeasTip(bExecute:= FALSE);
			IF pMzTool^.M_GetActionBusy(E_Action.ACTION_MoveXY) THEN
				pMzTool^.M_CancelAction(ACTION_MoveX);
				nActionState := 70;
			ELSIF pMzTool^.M_GetActionBusy(E_Action.ACTION_MoveZ) THEN
				pMzTool^.M_CancelAction(ACTION_MoveZ);
				nActionState := 70;
			ELSIF pMzTool^.P_pMzHead^.M_GetActionBusy(E_Action.ACTION_MoveZ) THEN
				pMzTool^.P_pMzHead^.M_CancelAction(ACTION_MoveZ);
				nActionState := 70;
			END_IF
		END_IF		
END_CASE

//Errorhandling
IF nActionState = 99 THEN
	fbMeasTip(bExecute:= FALSE);
	stError.ObjectId := pMzTool^.P_nObjectID;
	stError.Cmd := E_Action.ACTION_MeasureTool;
	stError.POUAction := E_POUACT.POUACT_A_MeasureTool;
	fbErrorList.M_Add(stError);
END_IF
END_ACTION

ACTION A_MeasureTipLegacy:
stError.POUState := nActionState;

IF pMzTool^.P_bError THEN
	stError.ErrorId := pMzTool^.P_nErrorId;
	nActionState := 99;
END_IF

CASE nActionState OF
	0:	//Alle Achsen des Heads auf Home fahren
		MEMSET(ADR(stActionData),0,SIZEOF(stActionData));
		stActionData.eAction := E_Action.ACTION_MoveZ;
		stActionData.aParams[1] := E_MoveMode.MODE_Home;
		stActionData.aParams[3] := -1;	//MaxSpeed Z
		stError.ErrorId := pMzTool^.P_pMzHead^.M_ExeAction(stActionData);
		IF stError.ErrorId > 0 THEN
			nActionState := 99;
		ELSE
			nActionState := 1;
		END_IF
		
	1:	//Head ready?
		IF NOT pMzTool^.P_pMzHead^.M_GetActionBusy(E_Action.ACTION_MoveZ) THEN
			IF pMzTool^.P_pMzHead^.P_bError THEN
				stError.ErrorId := pMzTool^.P_pMzHead^.P_nErrorId;
				nActionState := 99;
			ELSE
				nActionState := 2;
			END_IF
		END_IF	

	2:	//Vorberechnung und MoveXY(Startpos TipCalibrator)
		nActionState := 3;
	
		//Wenn noch nicht vermessen wurde und angeforderte Option = "MEAS_OPTION_OnlyXY", dann
		//Option auf "MEAS_OPTION_SlowApproach" ändern
		stPoint1 := pMzTool^.P_stRelPos;
		stPoint2 := pMzTool^.P_stOffset;
		
		//Wenn bisher noch nicht vermessen wurde, dann mit "SlowApproach" beginnen
		IF (NOT pMzTool^.P_bMeasured AND eMeasTipOption = E_MeasureOption.MEAS_OPTION_OnlyXY) OR (stPoint1.Z = 0 AND stPoint2.Z = 0) THEN
			eMeasTipOption := E_MeasureOption.MEAS_OPTION_SlowApproach;
		END_IF
		
		IF eMeasTipOption = E_MeasureOption.MEAS_OPTION_SlowApproach THEN
			IF pMzTool^.pPiece > 0 THEN
				pMzTool^.pPiece^.M_ClearOffset();
			ELSE
				pMzTool^.M_ClearOffset();	
			END_IF
		END_IF		
		
		//Startposition und Endposition des X-Moves berechnen
		stMeasPassIntersect := pTipCalibrator^.M_GetAbsPos(pChildPos:= 0, eTargetRef:= E_TargetRef.TARGETREF_SpecPoint,nParam1:= 1, nParam2:=0, nParam3:=0, nZLevel:=0);
		stMeasCalibPoint := pTipCalibrator^.M_GetAbsPos(pChildPos:= 0, eTargetRef:= E_TargetRef.TARGETREF_SpecPoint,nParam1:= 2, nParam2:=0, nParam3:=0, nZLevel:=0);
		stMeasStartPos := stMeasPassIntersect;
		stMeasStartPos.X := stMeasCalibPoint.X + rMeasureDistance;
		stMeasEndPos := stMeasPassIntersect;
		stMeasEndPos.X := stMeasCalibPoint.X - rMeasureDistance;
	
		//MoveXY auf stMeasStartPos
		MEMSET(ADR(stActionData),0,SIZEOF(stActionData));
		stActionData.eAction := E_Action.ACTION_MoveXY;
		stActionData.aParams[1] := E_MoveMode.MODE_AbsWithOffset;
		stActionData.aParams[2] := REAL_TO_DINT(stMeasStartPos.X); //XPos
		stActionData.aParams[3] := REAL_TO_DINT(stMeasStartPos.Y); //YPos
		stActionData.aParams[4] := -1;	//MaxSpeed X
		stActionData.aParams[5] := -1;	//MaxSpeed Y
		stError.ErrorId := pMzTool^.M_ExeAction(stActionData);
		IF stError.ErrorId > 0 THEN
			nActionState := 99;
		END_IF
		
	3:	//MoveXY ready? -> MoveZ auf StartPos
		IF NOT pMzTool^.M_GetActionBusy(E_Action.ACTION_MoveXY) THEN
			nActionState := 4;
			//ZMove auf stMeasStartPos
			MEMSET(ADR(stActionData),0,SIZEOF(stActionData));
			stActionData.eAction := E_Action.ACTION_MoveZ;
			stActionData.aParams[1] := E_MoveMode.MODE_AbsWithOffset;
			//In Abhängigkeit von MeasOption "Z" zustellen und Z-Feed voreinstellen
			CASE eMeasTipOption OF
				E_MeasureOption.MEAS_OPTION_SlowApproach: //keine Z-Zustellung, es von oben angefangen
					stActionData.aParams[1] := E_MoveMode.MODE_Home;
					fbMeasTip.nZFeedStart := -3000;
					fbMeasTip.nZFeedEnde := -50;
				E_MeasureOption.MEAS_OPTION_FastApproach:
					stActionData.aParams[1] := E_MoveMode.MODE_AbsWithOffset;
					fbMeasTip.nZFeedStart := -1000;
					fbMeasTip.nZFeedEnde := -50;
					fbMeasTip.nZFeedMax := -4000;
					stActionData.aParams[2] := REAL_TO_DINT(stMeasStartPos.Z); //ZPos
				E_MeasureOption.MEAS_OPTION_OnlyXY:
					stActionData.aParams[1] := E_MoveMode.MODE_AbsWithOffset;		
					stActionData.aParams[2] := REAL_TO_DINT(stMeasCalibPoint.Z) -300; //ZPos
			ELSE
				stError.ErrorId := E_ErrorIdCmd.ERRORID_InvalidMeasureMode;
			END_CASE
			
			IF stError.ErrorId > 0 THEN
				nActionState := 99;
			ELSE
				stActionData.aParams[3] := -1;	//MaxSpeed Z
				stError.ErrorId := pMzTool^.M_ExeAction(stActionData);
				IF stError.ErrorId > 0 THEN
					nActionState := 99;
				END_IF
			END_IF
		END_IF
		
	4:	//MoveZ ready?
		IF NOT pMzTool^.M_GetActionBusy(E_Action.ACTION_MoveZ) THEN
			IF pTipCalibrator^.P_bXSensor AND pTipCalibrator^.P_bYSensor THEN //Beide Lichtschranken müssen frei sein
				IF eMeasTipOption = E_MeasureOption.MEAS_OPTION_OnlyXY THEN
					nActionState := 11;
				ELSE
					IF eMeasTipOption = E_MeasureOption.MEAS_OPTION_SlowApproach THEN
						stPoint1 := pMzTool^.P_stCurrentPosPhys;
						stPoint2 := pTarget^.P_stAbsPosCenter;
						//der Kartuschenhalter kann so theoretisch bis 500µ über TipCalibrator heran 
						IF pMzTool^.P_pPiece > 0 THEN
							stDimension := pMzTool^.P_pPiece^.P_stDimension;
							fbMeasTip.nZFeedMax := - (REAL_TO_DINT(stPoint1.Z - stPoint2.Z + stDimension.Height - pMzTool^.P_pPiece^.P_rZOverlapTool) - 500);
						ELSE
							fbMeasTip.nZFeedMax := -(REAL_TO_DINT(stPoint1.Z - stPoint2.Z + 8500));
						END_IF
					END_IF
					nActionState := 5;	
				END_IF
			ELSE  //Error, mindestens eine der beiden Lichtschranken ist nicht frei
				stError.ErrorId := E_ErrorIdCmd.ERRORID_TipCalibSensor;
				nActionState := 99;
			END_IF 
		END_IF
		
	5:	//Z-Measurement
		fbMeasTip(bExecute:= TRUE, pMzTool:= pMzTool, pTipCalibrator:= pTipCalibrator, nDirection:= 3,
				 stStartPos:= stMeasStartPos, stEndPos:= stMeasEndPos);
	
		IF NOT fbMeasTip.bBusy THEN
			nActionState := 6;
			IF fbMeasTip.bError THEN //Error
				stError.ErrorId := fbMeasTip.nErrorId;
				nActionState := 99;
			ELSE
				//Gemessenen Z Wert verrechnen und als OffsetWert in Tool bzw Piece eintragen
				IF pMzTool^.pPiece > 0 THEN
					stMeasOffset := pMzTool^.pPiece^.P_stOffset;
					stMeasOffset.Z := stMeasOffset.Z - (fbMeasTip.stProbePos.Z - stMeasCalibPoint.Z);
					stMeasOffset.X := stMeasOffset.X - (fbMeasTip.stProbePos.X - stMeasCalibPoint.X);
					pMzTool^.pPiece^.P_stOffset := stMeasOffset;
				ELSE
					stMeasOffset := pMzTool^.P_stOffset;
					stMeasOffset.Z := stMeasOffset.Z - (fbMeasTip.stProbePos.Z - stMeasCalibPoint.Z);
					stMeasOffset.X := stMeasOffset.X - (fbMeasTip.stProbePos.X - stMeasCalibPoint.X);
					pMzTool^.P_stOffset := stMeasOffset;
				END_IF
				
				//Start und Endposition für folgende Y-Vermessung berechnen und in X auf Ausgangsposition fahren
				stMeasStartPos := stMeasPassIntersect;
				stMeasStartPos.Y := stMeasCalibPoint.Y - rMeasureDistance;
				stMeasEndPos := stMeasPassIntersect;
				stMeasEndPos.Y := stMeasCalibPoint.Y + rMeasureDistance;
				
				//MoveX StartPosX
				MEMSET(ADR(stActionData),0,SIZEOF(stActionData));
				stActionData.eAction := E_Action.ACTION_MoveX;
				stActionData.aParams[1] := E_MoveMode.MODE_AbsWithOffset;
				stActionData.aParams[2] := REAL_TO_DINT(stMeasStartPos.X); //XPos
				stActionData.aParams[3] := -1;	//MaxSpeed X
				stActionData.aParams[4] := 1; //ignore Z-Kollission
				stError.ErrorId := pMzTool^.M_ExeAction(stActionData);
				IF stError.ErrorId > 0 THEN //Error
					nActionState := 99;
				END_IF
			END_IF
			fbMeasTip(bExecute:= FALSE);	
		END_IF
		
	6:	//MoveX ready? -> MoveY StartPosY
		IF NOT pMzTool^.M_GetActionBusy(E_Action.ACTION_MoveX) THEN
			nActionState := 7;
			MEMSET(ADR(stActionData),0,SIZEOF(stActionData));
			stActionData.eAction := E_Action.ACTION_MoveY;
			stActionData.aParams[1] := E_MoveMode.MODE_AbsWithOffset;
			stActionData.aParams[2] := REAL_TO_DINT(stMeasStartPos.Y); //YPos
			stActionData.aParams[3] := -1;	//MaxSpeed Y
			stActionData.aParams[4] := 1; //ignore Z-Kollission
			stError.ErrorId := pMzTool^.M_ExeAction(stActionData);		
			IF stError.ErrorId > 0 THEN //Error
				nActionState := 99;
			END_IF
		END_IF
		
	7:	//MoveY ready? -> MoveZ auf StartPointZ (300µ unterhalb CalibPoint)
		IF NOT pMzTool^.M_GetActionBusy(E_Action.ACTION_MoveY) THEN
			nActionState := 8;
			MEMSET(ADR(stActionData),0,SIZEOF(stActionData));
			stActionData.eAction := E_Action.ACTION_MoveZ;
			stActionData.aParams[1] := E_MoveMode.MODE_AbsWithOffset;
			stActionData.aParams[2] := REAL_TO_DINT(stMeasCalibPoint.Z) -300;
			stActionData.aParams[3] := -1;	//MaxSpeed Z
			stError.ErrorId := pMzTool^.M_ExeAction(stActionData); //ErrorHandling am Ende
			IF stError.ErrorId > 0 THEN //Error
				nActionState := 99;
			END_IF
		END_IF

	8:	//MoveZ ready? -> weiter zu Y-Measurement
		IF NOT pMzTool^.M_GetActionBusy(E_Action.ACTION_MoveZ) THEN
			nActionState := 9;
		END_IF
		
	9:	//Y-Measurement
		fbMeasTip(bExecute:= TRUE, pMzTool:= pMzTool, pTipCalibrator:= pTipCalibrator, nDirection:= 2,
					stStartPos:= stMeasStartPos, stEndPos:= stMeasEndPos);		
	
		IF NOT fbMeasTip.bBusy THEN
			IF fbMeasTip.bError THEN
				stError.ErrorId := fbMeasTip.nErrorId;
				nActionState := 99;
			ELSE
				//Gemessenen Y Wert verrechnen und als OffsetWert in Tool eintragen
				IF pMzTool^.pPiece > 0 THEN
					stMeasOffset := pMzTool^.pPiece^.P_stOffset;
					stMeasOffset.Y := stMeasOffset.Y - (fbMeasTip.stProbePos.Y - stMeasCalibPoint.Y);
					pMzTool^.pPiece^.P_stOffset := stMeasOffset;
				ELSE
					stMeasOffset := pMzTool^.P_stOffset;
					stMeasOffset.Y := stMeasOffset.Y - (fbMeasTip.stProbePos.Y - stMeasCalibPoint.Y);
					pMzTool^.P_stOffset := stMeasOffset;
				END_IF				
				
				//Start und Endposition für folgende Y-Vermessung berechnen und in X auf Ausgangsposition fahren
				stMeasStartPos := stMeasPassIntersect;
				stMeasStartPos.X := stMeasCalibPoint.X + rMeasureDistance;
				stMeasEndPos := stMeasPassIntersect;
				stMeasEndPos.X := stMeasCalibPoint.X - rMeasureDistance;
				
				IF eMeasTipOption = E_MeasureOption.MEAS_OPTION_OnlyXY THEN
					//Z-Achse freifahren
					MEMSET(ADR(stActionData),0,SIZEOF(stActionData));
					stActionData.eAction := E_Action.ACTION_MoveZ;
					stActionData.aParams[1] := E_MoveMode.MODE_Free;
					stActionData.aParams[3] := -1;	//MaxSpeed Z
					stError.ErrorId := pMzTool^.M_ExeAction(stActionData);
					IF stError.ErrorId > 0 THEN //Error
						nActionState := 99;
					ELSE
						nActionState := 12;	
					END_IF
				ELSE
					MEMSET(ADR(stActionData),0,SIZEOF(stActionData));
					stActionData.eAction := E_Action.ACTION_MoveY;
					stActionData.aParams[1] := E_MoveMode.MODE_AbsWithOffset;
					stActionData.aParams[2] := REAL_TO_DINT(stMeasStartPos.Y); //YPos
					stActionData.aParams[3] := -1;	//MaxSpeed Y
					stActionData.aParams[4] := 1; //ignore Z-Kollission
					stError.ErrorId := pMzTool^.M_ExeAction(stActionData);
					IF stError.ErrorId > 0 THEN //Error
						nActionState := 99;
					ELSE
						nActionState := 10;	
					END_IF
				END_IF
			END_IF
			fbMeasTip(bExecute:= FALSE);	
		END_IF
		
	10:	//MoveY ready?
		IF NOT pMzTool^.M_GetActionBusy(E_Action.ACTION_MoveY) THEN
			nActionState := 11;
		END_IF
		
	11:	//X-Measurement
		fbMeasTip(bExecute:= TRUE, pMzTool:= pMzTool, pTipCalibrator:= pTipCalibrator, nDirection:= 1,
					stStartPos:= stMeasStartPos, stEndPos:= stMeasEndPos);
					
		IF NOT fbMeasTip.bBusy THEN
			IF fbMeasTip.bError THEN
				stError.ErrorId := fbMeasTip.nErrorId;
			ELSE
				//Wenn Piece am Tool, den Offset des Pieces verrechnen sonst des Tools
				IF pMzTool^.pPiece > 0 THEN
					stMeasOffset := pMzTool^.pPiece^.P_stOffset;
					stMeasOffset.X := stMeasOffset.X - (fbMeasTip.stProbePos.X - stMeasCalibPoint.X);
					pMzTool^.pPiece^.P_stOffset := stMeasOffset;
				ELSE
					stMeasOffset := pMzTool^.P_stOffset;
					stMeasOffset.X := stMeasOffset.X - (fbMeasTip.stProbePos.X - stMeasCalibPoint.X);
					pMzTool^.P_stOffset := stMeasOffset;
				END_IF
				
				IF eMeasTipOption = E_MeasureOption.MEAS_OPTION_OnlyXY THEN
					//weiter zu Y-Vermessung
					//Start und Endposition für folgende Y-Vermessung berechnen und in X auf Ausgangsposition fahren
					stMeasStartPos := stMeasPassIntersect;
					stMeasStartPos.Y := stMeasCalibPoint.Y - rMeasureDistance;
					stMeasEndPos := stMeasPassIntersect;
					stMeasEndPos.Y := stMeasCalibPoint.Y + rMeasureDistance;
					
					MEMSET(ADR(stActionData),0,SIZEOF(stActionData));
					stActionData.eAction := E_Action.ACTION_MoveX;
					stActionData.aParams[1] := E_MoveMode.MODE_AbsWithOffset;
					stActionData.aParams[2] := REAL_TO_DINT(stMeasStartPos.X); //XPos
					stActionData.aParams[3] := -1;	//MaxSpeed X
					stActionData.aParams[4] := 1; //ignore Z-Kollission
					stError.ErrorId := pMzTool^.M_ExeAction(stActionData);
					IF stError.ErrorId > 0 THEN //Error
						nActionState := 99;
					ELSE
						nActionState := 6;	
					END_IF
				ELSE
					//MoveZ-Free
					MEMSET(ADR(stActionData),0,SIZEOF(stActionData));
					stActionData.eAction := E_Action.ACTION_MoveZ;
					stActionData.aParams[1] := E_MoveMode.MODE_Free;
					stActionData.aParams[3] := -1;	//MaxSpeed Z
					stError.ErrorId := pMzTool^.M_ExeAction(stActionData);
					IF stError.ErrorId > 0 THEN //Error
						nActionState := 99;
					ELSE
						nActionState := 12;	
					END_IF
				END_IF
			END_IF
			fbMeasTip(bExecute:= FALSE);
		END_IF					
	
	12:	//MoveZ-Free ready? -> Action ready
		IF NOT pMzTool^.M_GetActionBusy(E_Action.ACTION_MoveZ) THEN
			IF pMzTool^.P_pPiece > 0 THEN
				fbObjectDirectory.M_SetObjChange(pMzTool^.pPiece^.P_nObjectID);
			ELSE
				fbObjectDirectory.M_SetObjChange(pMzTool^.P_nObjectID);
			END_IF			
			pMzTool^.P_bMeasured := TRUE;
			nActionState := 80;
		END_IF
	
	70:	//Action abbrechen
		nActionState := 80;
		IF fbMeasTip.bBusy THEN
			fbMeasTip.M_Cancel();
			fbMeasTip();
			nActionState := 70;
		ELSE
			fbMeasTip(bExecute:= FALSE);
			IF pMzTool^.M_GetActionBusy(E_Action.ACTION_MoveX) THEN
				pMzTool^.M_CancelAction(ACTION_MoveX);
				nActionState := 70;
			ELSIF pMzTool^.M_GetActionBusy(E_Action.ACTION_MoveY) THEN
				pMzTool^.M_CancelAction(ACTION_MoveY);
				nActionState := 70;
			ELSIF pMzTool^.M_GetActionBusy(E_Action.ACTION_MoveXY) THEN
				pMzTool^.M_CancelAction(ACTION_MoveXY);
				nActionState := 70;
			ELSIF pMzTool^.M_GetActionBusy(E_Action.ACTION_MoveZ) THEN
				pMzTool^.M_CancelAction(ACTION_MoveZ);
				nActionState := 70;				
			END_IF
		END_IF
END_CASE

//Errorhandling
IF nActionState = 99 THEN
	fbMeasTip(bExecute:= FALSE);
	stError.ObjectId := pMzTool^.P_nObjectID;
	stError.Cmd := E_Action.ACTION_MeasureTool;
	stError.POUAction := E_POUACT.POUACT_A_MeasureTool;
	fbErrorList.M_Add(stError);
END_IF
END_ACTION

ACTION A_MoveAllHome:
stError.POUState := nActionState;

CASE nActionState OF
	0:	//MoveZ Heads in Home
		MEMSET(ADR(stActionData),0,SIZEOF(stActionData));
		stActionData.eAction := E_Action.ACTION_MoveZ;
		stActionData.aParams[1] := E_MoveMode.MODE_Home;
		stActionData.aParams[3] := -1;
		nActionState := 1;
		FOR i:= 1 TO fbObjectDirectory.nCntMZHead BY 1 DO
			stError.ErrorId := afbMzHead[i].M_ExeAction(stActionData);
			IF stError.ErrorId > 0 THEN
				stError.HardwareGrp := E_HardwareGrp.AxisZ;
				stError.HardwareNr := 0;
				nActionState := 99;
				EXIT;
			END_IF
		END_FOR
		
	1:	//Alle Heads fertig?
		nActionState := 2;
		FOR i:= 1 TO fbObjectDirectory.nCntMZHead BY 1 DO
			IF afbMzHead[i].P_bError THEN
				stError.ErrorId := afbMzHead[i].P_nErrorId;
				nActionState := 99;
				EXIT;
			ELSIF afbMzHead[i].M_GetActionBusy(E_Action.ACTION_MoveZ) THEN
				nActionState := 1;
				EXIT;
			END_IF
		END_FOR
		
	2:	//Heads in X und Y in max Pos fahren
		//In X braucht nur der erste Head fahren, da der zweite (wenn vorhanden) ja an der gleiche X-Achse hängt
		nActionState := 3;
		MEMSET(ADR(stActionData),0,SIZEOF(stActionData));
		stActionData.eAction := E_Action.ACTION_MoveXY;
		stActionData.aParams[1] := E_MoveMode.MODE_AbsNoneOffset;
		stActionData.aParams[2] :=  REAL_TO_DINT(afbMzHead[1].P_pXDrive^.P_rMaxPos);
		stActionData.aParams[3] :=  REAL_TO_DINT(afbMzHead[1].P_pYDrive^.P_rMaxPos);
		stActionData.aParams[4] :=  -1;
		stActionData.aParams[5] :=  -1;
		stError.ErrorId := afbMzHead[1].M_ExeAction(stActionData);
		
		IF stError.ErrorId = 0 THEN
			{IF defined (TwoHeads)}
			IF afbMzHead[2].P_nObjectID > 0 THEN	//zweiter Head vorhanden
				stActionData.eAction := E_Action.ACTION_MoveY;
				stActionData.aParams[2] :=  REAL_TO_DINT(afbMzHead[2].P_pYDrive^.P_rMaxPos);
				stActionData.aParams[3] :=  -1;
				stError.ErrorId := afbMzHead[2].M_ExeAction(stActionData);
				IF stError.ErrorId > 0 THEN
					stError.HardwareGrp := E_HardwareGrp.AxisY;
					stError.HardwareNr := 0;
					nActionState := 99;
				END_IF
			END_IF
			{END_IF}
		ELSE
			stError.HardwareGrp := E_HardwareGrp.AxisX;
			stError.HardwareNr := 0;
			nActionState := 99;
		END_IF
		
	3:	//Alle Heads fertig?
		nActionState := 80;
		FOR i:= 1 TO fbObjectDirectory.nCntMZHead BY 1 DO
			IF afbMzHead[i].P_bError THEN
				stError.ErrorId := afbMzHead[i].P_nErrorId;
				nActionState := 99;
				EXIT;
			ELSIF afbMzHead[i].M_GetActionBusy(E_Action.ACTION_MoveXY) THEN
				nActionState := 3;
				EXIT;
			END_IF
		END_FOR
		
	70:	//Heads
		FOR i:= 1 TO fbObjectDirectory.nCntMZHead BY 1 DO
			afbMzHead[i].M_Stop();
		END_FOR
		nActionState := 71;
		
	71:	//Heads gestoppt?
		nActionState := 80;
		FOR i:= 1 TO fbObjectDirectory.nCntMZHead BY 1 DO
			IF afbMzHead[i].bBusy THEN
				nActionState := 71;
			END_IF
		END_FOR
		
END_CASE

//Errorhandling
IF nActionState = 99 THEN
	stError.Cmd := E_Action.ACTION_MoveAllHome;
	stError.POUAction := E_POUACT.POUACT_A_MoveAllHome;
	fbErrorList.M_Add(stError);
END_IF
END_ACTION

ACTION A_MoveToTarget:
stError.POUState := nActionState;

IF nActionState = 0 THEN
	fbMoveToTarget(bExecute:= TRUE);
	IF NOT fbMoveToTarget.bBusy THEN
		IF fbMoveToTarget.bError THEN
			stError.ErrorId := fbMoveToTarget.nErrorId;
			nActionState := 99;
		ELSE
			nActionState := 80;
		END_IF
		fbMoveToTarget(bExecute:= FALSE);
	END_IF
ELSIF nActionState = 70 THEN	//Abbrechen
	IF fbMoveToTarget.bBusy THEN
		fbMoveToTarget(bStop:= TRUE);
	ELSE	
		fbMoveToTarget(bExecute:= FALSE);
		nActionState := 80;
	END_IF
END_IF


//Errorhandling
IF nActionState = 99 THEN
	//stError.ObjectId := 
	stError.Cmd := E_Action.ACTION_MoveToTarget;
	stError.POUAction := E_POUACT.POUACT_A_MoveToTarget;
	fbErrorList.M_Add(stError);
END_IF
END_ACTION

ACTION A_OpenCloseFlipTube:
stError.POUState := nActionState;

IF pMzTool^.P_bError THEN
	stError.ObjectId := pMzTool^.P_nObjectID;
	stError.ErrorId := pMzTool^.P_nErrorId;
	nActionState := 99;
END_IF

IF pMzTool^.P_bCanceled AND nActionState > 0 AND nActionState < 70 THEN
	//MzTool wurde durch StopDevice abgebrochen
	nActionState := 70;
END_IF

CASE nActionState OF
	0:	//MoveToTarget auf Slot
		MEMSET(ADR(stActionData),0,SIZEOF(stActionData));
		stActionData.eAction := E_Action.ACTION_MoveToTarget;
		stActionData.nObject := pMzTool^.P_nObjectID;
		stActionData.nTarget := pTarget^.P_nObjectID;
		stActionData.aParams[1] := E_TargetRef.TARGETREF_Slot;
		stActionData.aParams[2] := pPieceSlot^.nNr;
		stActionData.aParams[3] := 0;
		stActionData.aParams[5] := -1;	//MaxSpeed X
		stActionData.aParams[6] := -1;	//MaxSpeed Y
		stActionData.aParams[7] := -1;	//MaxSpeed Z
		IF bOpen THEN
			stPoint1 := pFlipTubeRack^.P_stOpenStartPos;
		ELSE
			stPoint1 := pFlipTubeRack^.P_stCloseStartPos;
		END_IF
		stActionData.aParams[8] := REAL_TO_DINT(stPoint1.X);
		stActionData.aParams[9] := REAL_TO_DINT(stPoint1.Y);
		stActionData.aParams[10] := REAL_TO_DINT(stPoint1.Z);
		stError.ErrorId := fbMoveToTarget.M_SetAndCheckParams(stActionData);
		IF stError.ErrorId > 0 THEN	//Error
			nActionState := 99;
		ELSE
			fbMoveToTarget(bExecute:= TRUE);
			nActionState := 1;
		END_IF		

	1:	//MoveToTarget ready? -> "Open Move1" bzw. "Close Move1"
		fbMoveToTarget(bExecute:= TRUE);
		IF NOT fbMoveToTarget.bBusy THEN
			IF fbMoveToTarget.bError THEN
				stError.ErrorId := fbMoveToTarget.nErrorId;
			ELSE
				pFlipTube := pPieceSlot^.P_pPiece;
				IF bOpen THEN
					nActionState := 2;
				ELSE
					nActionState := 10;
				END_IF
			END_IF
			fbMoveToTarget(bExecute:= FALSE);
		END_IF	
		
	2:	//Open Move1 (Z)
		nActionState := 3;
		MEMSET(ADR(stActionData),0,SIZEOF(stActionData));
		stActionData.eAction := E_Action.ACTION_MoveZ;
		stActionData.aParams[1] := E_MoveMode.MODE_Relative;
		stActionData.aParams[2] := pFlipTubeRack^.P_nOpenMove1DistZ;
		stActionData.aParams[3] := 2000; //SpeedZ
		stError.ErrorId := pMzTool^.M_ExeAction(stActionData);
		IF stError.ErrorId > 0 THEN	//Error
			nActionState := 99;
		END_IF
			
	3:	//Open Move2 (Z)
		IF NOT pMzTool^.M_GetActionBusy(E_Action.ACTION_MoveZ) THEN
			nActionState := 4;
			MEMSET(ADR(stActionData),0,SIZEOF(stActionData));
			stActionData.eAction := E_Action.ACTION_MoveZ;
			stActionData.aParams[1] := E_MoveMode.MODE_Relative;
			stActionData.aParams[2] := pFlipTubeRack^.P_nOpenMove2DistZ;
			stActionData.aParams[3] := -1; //SpeedZ
			stError.ErrorId := pMzTool^.M_ExeAction(stActionData);
			IF stError.ErrorId > 0 THEN	//Error
				nActionState := 99;
			END_IF
		END_IF
	
	4:	//Open Move3 (Y)
		IF NOT pMzTool^.M_GetActionBusy(E_Action.ACTION_MoveZ) THEN
			nActionState := 5;
			MEMSET(ADR(stActionData),0,SIZEOF(stActionData));
			stActionData.eAction := E_Action.ACTION_MoveY;
			stActionData.aParams[1] := E_MoveMode.MODE_Relative;
			stActionData.aParams[2] := pFlipTubeRack^.P_nOpenMove3DistY;
			stActionData.aParams[3] := -1; //SpeedY
			stActionData.aParams[4] := 1; //IgnoreZCollision
			stError.ErrorId := pMzTool^.M_ExeAction(stActionData);
			IF stError.ErrorId > 0 THEN	//Error
				nActionState := 99;
			END_IF
		END_IF
		
	5:	//Open Move4 (X)
		IF NOT pMzTool^.M_GetActionBusy(E_Action.ACTION_MoveY) THEN
			nActionState := 6;
			MEMSET(ADR(stActionData),0,SIZEOF(stActionData));
			stActionData.eAction := E_Action.ACTION_MoveX;
			stActionData.aParams[1] := E_MoveMode.MODE_Relative;
			stActionData.aParams[2] := pFlipTubeRack^.P_nOpenMove4DistX;
			stActionData.aParams[3] := -1; //SpeedX
			stActionData.aParams[4] := 1; //IgnoreZCollision
			stError.ErrorId := pMzTool^.M_ExeAction(stActionData);
			IF stError.ErrorId > 0 THEN	//Error
				nActionState := 99;
			END_IF
		END_IF		
	
	6:	//Open Move4 -> letzter Z-Move
		IF NOT pMzTool^.M_GetActionBusy(E_Action.ACTION_MoveX) THEN
			MEMSET(ADR(stActionData),0,SIZEOF(stActionData));
			stActionData.eAction := E_Action.ACTION_MoveZ;
			stActionData.aParams[1] := E_MoveMode.MODE_Relative;
			stActionData.aParams[2] := pFlipTubeRack^.P_nOpenMove5DistZ;
			stActionData.aParams[3] := 20000; //SpeedZ
			stError.ErrorId := pMzTool^.M_ExeAction(stActionData);
			IF stError.ErrorId > 0 THEN	//Error
				nActionState := 99;
			ELSE
				nActionState := 20;
				pFlipTube^.P_bIsOpen := TRUE;	
			END_IF
		END_IF
		
	10: //Close Move1
		MEMSET(ADR(stActionData),0,SIZEOF(stActionData));
		stActionData.eAction := E_Action.ACTION_MoveX;
		stActionData.aParams[1] := E_MoveMode.MODE_Relative;
		stActionData.aParams[2] := pFlipTubeRack^.P_nCloseMove1DistX;
		stActionData.aParams[3] := 45000; //SpeedX
		stActionData.aParams[4] := 1; //IgnoreZCollision
		stError.ErrorId := pMzTool^.M_ExeAction(stActionData);
		IF stError.ErrorId > 0 THEN	//Error
			nActionState := 99;
		ELSE
			nActionState := 11;
		END_IF
	
	11: //Close Move2 -> letzter Z-Move
		IF NOT pMzTool^.M_GetActionBusy(E_Action.ACTION_MoveX) THEN
			MEMSET(ADR(stActionData),0,SIZEOF(stActionData));
			stActionData.eAction := E_Action.ACTION_MoveZ;
			stActionData.aParams[1] := E_MoveMode.MODE_Relative;
			stActionData.aParams[2] := pFlipTubeRack^.P_nCloseMove2DistZ;
			stActionData.aParams[3] := 2000; //SpeedZ
			stError.ErrorId := pMzTool^.M_ExeAction(stActionData);
			IF stError.ErrorId > 0 THEN	//Error
				nActionState := 99;
			ELSE
				nActionState := 20;
				pFlipTube^.P_bIsOpen := FALSE;
			END_IF
		END_IF
	
	20:	//MoveZ
		IF NOT pMzTool^.M_GetActionBusy(E_Action.ACTION_MoveZ) THEN
			MEMSET(ADR(stActionData),0,SIZEOF(stActionData));
			stActionData.eAction := E_Action.ACTION_MoveZ;
			stActionData.aParams[1] := E_MoveMode.MODE_Free;
			stError.ErrorId := pMzTool^.M_ExeAction(stActionData);
			IF stError.ErrorId > 0 THEN	//Error
				nActionState := 99;
			ELSE
				nActionState := 21;
			END_IF
		END_IF
		
	21:	//MoveZ-Free ready?
		IF NOT pMzTool^.M_GetActionBusy(E_Action.ACTION_MoveZ) THEN
			fbObjectDirectory.M_SetObjChange(pFlipTube^.P_nObjectID);
			nActionState := 80;
		END_IF
	
	70:	//Abbrechen
		IF fbMoveToTarget.bBusy THEN
			fbMoveToTarget(bStop:= TRUE);
		ELSIF pMzTool^.M_GetActionBusy(E_Action.ACTION_MoveX) THEN
			pMzTool^.M_CancelAction(E_Action.ACTION_MoveX);
		ELSIF pMzTool^.M_GetActionBusy(E_Action.ACTION_MoveY) THEN
			pMzTool^.M_CancelAction(E_Action.ACTION_MoveY);
		ELSIF pMzTool^.M_GetActionBusy(E_Action.ACTION_MoveZ) THEN
			pMzTool^.M_CancelAction(E_Action.ACTION_MoveZ);
		ELSE
			fbMoveToTarget(bExecute:= FALSE);
			nActionState := 80;
		END_IF
END_CASE

//Errorhandling
IF nActionState = 99 THEN
	fbMoveToTarget(bExecute:= FALSE);
	stError.ObjectId := pMzTool^.P_nObjectID;
	stError.Cmd := E_Action.ACTION_OpenCloseFlipTube;
	stError.POUAction := E_POUACT.POUACT_A_OpenCloseFlipTube;
	fbErrorList.M_Add(stError);
END_IF
END_ACTION

ACTION A_StampDemold:
stError.POUState := nActionState;

IF pMzTool^.P_bError THEN
	stError.ErrorId := pMzTool^.P_nErrorId;
	nActionState := 99;
END_IF

IF pMzTool^.P_bCanceled AND nActionState > 0 AND nActionState < 70 THEN
	//MzTool wurde durch StopDevice abgebrochen
	nActionState := 70;
END_IF

CASE nActionState OF
	0:	//Set Pressure
		nActionState := 1;
		stActionData.eAction := E_Action.ACTION_SetPressure;
		stActionData.aParams[1] := 1;
		stActionData.aParams[2] := nPressure1;
		stActionData.aParams[3] := 5;	//Tolerance +
		stActionData.aParams[4] := 5;	//Tolerance -
		stActionData.aParams[5] := 2000;	//Timeout
		stError.ErrorId := pStampSupport^.M_ExeAction(stActionData);
		IF stError.ErrorId > 0 THEN
			nActionState := 99;
		END_IF

	1:	//Pressure ready?
 		IF NOT pStampSupport^.M_GetActionBusy(E_Action.ACTION_SetPressure) THEN
			nActionState := 2;
		END_IF
		
	2:	//Set Vacuum
		nActionState := 3;
		stActionData.eAction := E_Action.ACTION_SetVacuum;
		stActionData.aParams[1] := 1;
		stActionData.aParams[2] := nPressure2;
		stActionData.aParams[3] := 5;	//Tolerance +
		stActionData.aParams[4] := 5;	//Tolerance -
		stActionData.aParams[5] := 2000;	//Timeout
		stError.ErrorId := pStampSupport^.M_ExeAction(stActionData);
		IF stError.ErrorId > 0 THEN
			nActionState := 99;
		END_IF
		
	3:	//Vacuum ready?
 		IF NOT pStampSupport^.M_GetActionBusy(E_Action.ACTION_SetVacuum) THEN
			nActionState := 4;
		END_IF
		
	4:	//MoveZ
		nActionState := 5;
		MEMSET(ADR(stActionData),0,SIZEOF(stActionData));
		stActionData.eAction := E_Action.ACTION_MoveZ;
		stActionData.aParams[1] := E_MoveMode.MODE_Relative;
		stActionData.aParams[2] := nDistance1;
		stActionData.aParams[3] := nSpeed1;
		stError.ErrorId := pStampSupport^.M_ExeAction(stActionData);
		IF stError.ErrorId > 0 THEN
			nActionState := 99;
		END_IF
		
	5:	//PulsePressure
		nActionState := 6;
		//stActionData.bIntern := TRUE;
		stActionData.eAction := E_Action.ACTION_PulsePressure;
		stActionData.aParams[1] := E_PressCtrl.PRESSCTRL_VacOn;	//Phase 1
		stActionData.aParams[2] := E_PressCtrl.PRESSCTRL_PressOn;	//Phase 2
		stActionData.aParams[3] := nPeriode;
		stActionData.aParams[4] := nDutycycle;
		stActionData.aParams[5] := 0;	//Dauerpulsen
		stActionData.aParams[6] := 1;	//On
		stError.ErrorId := pStampSupport^.M_ExeAction(stActionData);
		IF stError.ErrorId > 0 THEN
			nActionState := 99;
		END_IF		
		
	6:	//MoveZ ready? -> PulsePressure off
 		IF NOT pStampSupport^.M_GetActionBusy(E_Action.ACTION_MoveZ) THEN
			nActionState := 7;
			stActionData.aParams[6] := 0;	//PulsePressure Off
			stError.ErrorId := pStampSupport^.M_ExeAction(stActionData);
			IF stError.ErrorId > 0 THEN
				nActionState := 99;
			END_IF			
		END_IF
		
	7:	//PulsePressure ready? -> Action ready
 		IF NOT pStampSupport^.M_GetActionBusy(E_Action.ACTION_PulsePressure) THEN
			nActionState := 80;
		END_IF
		
	70:	//Abbrechen
		nActionState := 80;
		IF pStampSupport^.M_GetActionBusy(E_Action.ACTION_SetPressure) THEN
			pStampSupport^.M_CancelAction(E_Action.ACTION_SetPressure);
			nActionState := 70;
		END_IF

		IF pStampSupport^.M_GetActionBusy(E_Action.ACTION_SetVacuum) THEN
			pStampSupport^.M_CancelAction(E_Action.ACTION_SetVacuum);
			nActionState := 70;
		END_IF
		
		IF pStampSupport^.M_GetActionBusy(E_Action.ACTION_PulsePressure) THEN
			pStampSupport^.M_CancelAction(E_Action.ACTION_PulsePressure);
			nActionState := 70;
		END_IF
		
		IF pStampSupport^.M_GetActionBusy(E_Action.ACTION_MoveZ) THEN
			pStampSupport^.M_CancelAction(E_Action.ACTION_MoveZ);
			nActionState := 70;
		END_IF
		
END_CASE

//Errorhandling
IF nActionState = 99 THEN
	stError.ObjectId := pMzTool^.P_nObjectID;
	stError.Cmd := E_Action.ACTION_StampDemolding;
	stError.POUAction := E_POUACT.POUACT_A_StampDemold;
	fbErrorList.M_Add(stError);
END_IF
END_ACTION

ACTION A_StampInking:
stError.POUState := nActionState;
IF pInkStation > 0 AND_THEN pInkStation^.P_bError THEN
	stError.ErrorId := pInkStation^.P_nErrorId;
	stError.ObjectId := pTarget^.P_nObjectID;
	nActionState := 99;
ELSIF pStampSupport^.P_bError THEN
	stError.ErrorId := pStampSupport^.P_nErrorId;
	stError.ObjectId := pStampSupport^.P_nObjectID;
	nActionState := 99;	
END_IF

IF pStampSupport^.P_bCanceled AND nActionState > 0 AND nActionState < 70 THEN
	//MzTool wurde durch StopDevice abgebrochen
	nActionState := 70;
END_IF

CASE nActionState OF
	0:	
		IF pInkStation = 0 THEN
			nActionState := 2;
			RETURN;
		END_IF
		nActionState := 1;
		//Wenn noch Spinning, dann anhalten
		IF pInkStation^.P_bIsSpinning THEN
			stActionData.eAction := E_Action.ACTION_InkSpin;
			stActionData.aParams[1] := 0;
			stActionData.aParams[2] := 0;
			stError.ErrorId := pInkStation^.M_ExeAction(stActionData);
			IF stError.ErrorId > 0 THEN
				stError.ObjectId := pTarget^.P_nObjectID;
				nActionState := 99;
			END_IF
		END_IF
	
	1:	//Wenn Deckel geschlossen, dann öffnen
		nActionState := 2;
		IF pInkStation^.P_eCoverState <> E_OpClState.Open THEN
			stActionData.eAction := E_Action.ACTION_InkOpClCover;
			stActionData.aParams[1] := 0;
			stError.ErrorId := pInkStation^.M_ExeAction(stActionData);
			IF stError.ErrorId > 0 THEN
				stError.ObjectId := pTarget^.P_nObjectID;
				nActionState := 99;
			END_IF
		END_IF
	
	2:	//Wenn Druck auf Stempel, dann Druck aus
		IF pStampSupport^.P_eCurPressState <> E_PressCtrl.PRESSCTRL_Off THEN
			stActionData.eAction := E_Action.ACTION_SwitchPressure;
			stActionData.aParams[1] := E_PressCtrl.PRESSCTRL_Off; 
			stError.ErrorId := pStampSupport^.M_ExeAction(stActionData);
			IF stError.ErrorId > 0 THEN
				stError.ObjectId := pStampSupport^.P_nObjectID;
				nActionState := 99;
			END_IF
		ELSE
			//Druck voreinstellen
			stActionData.eAction := E_Action.ACTION_SetPressure;
			stActionData.aParams[1] := 0;	//Action wird sofort fertig gemeldet
 			stActionData.aParams[2] := nPressure1;
			stError.ErrorId := pStampSupport^.M_ExeAction(stActionData);
			IF stError.ErrorId > 0 THEN
				stError.ObjectId := pStampSupport^.P_nObjectID;
				nActionState := 99;
			ELSE
				nActionState := 3;	
			END_IF
		END_IF
		
	3:	//Target eine InkStation? Open?
		nActionState := 4;
		IF pInkStation > 0 THEN
			IF NOT pInkStation^.M_GetActionBusy(E_Action.ACTION_InkOpClCover) THEN
				IF pInkStation^.P_eCoverState <> E_OpClState.Open THEN //Error
					stError.ObjectId := pInkStation^.P_nObjectID;
					stError.ErrorId := E_ErrorIdCmd.ERRORID_InkStationNotOpen;
					nActionState := 99;
				END_IF
			ELSE
				nActionState := 3;
			END_IF
		END_IF
	
	4:	//MoveToTarget
		MEMSET(ADR(stActionData),0,SIZEOF(stActionData));
		stActionData.eAction := E_Action.ACTION_MoveToTarget;
		stActionData.nObject := pStampSupport^.P_nObjectID;
		stActionData.nTarget := pTarget^.P_nObjectID;
		IF pInkStation > 0 THEN	//Inkstation
			stActionData.aParams[1] := E_TargetRef.TARGETREF_SpecPoint;
			stActionData.aParams[2] := 2; //Inkpoint
		ELSE //Point
			stActionData.aParams[1] := E_TargetRef.TARGETREF_Center;
		END_IF
		stActionData.aParams[5] := -1;	//MaxSpeed X
		stActionData.aParams[6] := -1;	//MaxSpeed Y
		stActionData.aParams[7] := -1;	//MaxSpeed Z
		stActionData.aParams[10] := nDistance1;
		stError.ErrorId := fbMoveToTarget.M_SetAndCheckParams(stActionData);
		IF stError.ErrorId > 0 THEN	//Error
			stError.ObjectId := pStampSupport^.P_nObjectID;
			nActionState := 99;
		ELSE
			fbMoveToTarget(bExecute:= TRUE);
			nActionState := 5;
		END_IF
	
